(* ToolTens force +,++,-,-- *)
	IF xToolTensForceAdd OR xToolTensForceAddMore OR xToolTensForceSub OR xToolTensForceSubMore THEN
		CASE iStepAction OF
		(* check cylinder state *)
		1:	xTmp:=	ptrCylAction^.T_CtrleCyl.xDone
					AND NOT(ptrCylAction^.T_CtrleCyl.xExecute)
					AND NOT(ptrCylAction^.T_CtrleCyl.xErr)
					AND ptrCylAction^.T_CtrleCyl.T_AnalogCylinder.xActiv;
			(* next step *)
			IF xTmp THEN iStepAction:=10; ELSE iStepAction:=95; END_IF
			IF xTmp AND T_Station.TControl.xHardwareConfigError THEN iStepAction:=95; END_IF;
		10:	IF xToolTensForceAdd THEN
				rCorrectionValue:=0.1;
			END_IF;
			IF xToolTensForceAddMore THEN
				rCorrectionValue:=1.0;
			END_IF;
			IF xToolTensForceSub THEN
				rCorrectionValue:=-0.1;
			END_IF;
			IF xToolTensForceSubMore THEN
				rCorrectionValue:=-1.0;
			END_IF;
			T_Visu.ptrT_ExchgParam^.T_InfoValueCommon.rToolTensionForce:=T_Visu.ptrT_ExchgParam^.T_InfoValueCommon.rToolTensionForce + rCorrectionValue;
			IF (T_Visu.ptrT_ExchgParam^.T_InfoValueCommon.rToolTensionForce < 0.1) THEN
				T_Visu.ptrT_ExchgParam^.T_InfoValueCommon.rToolTensionForce:=0.0;
			END_IF;
			IF (T_Visu.ptrT_ExchgParam^.T_InfoValueCommon.rToolTensionForce > T_NovRAM.T_Data.T_Standard.T_ToolTensionSystem.rMaxForceTT) THEN
				T_Visu.ptrT_ExchgParam^.T_InfoValueCommon.rToolTensionForce:=T_NovRAM.T_Data.T_Standard.T_ToolTensionSystem.rMaxForceTT;
			END_IF;
			(* next step *)
			iStepAction:=20;
		(* activ function set analog value *)
		20:	ptrCylAction^.T_CtrleCyl.T_AnalogCylinder.rForceIn:=T_Visu.ptrT_ExchgParam^.T_InfoValueCommon.rToolTensionForce;
			ptrCylAction^.T_CtrleCyl.iFunction:=4;
			ptrCylAction^.T_CtrleCyl.xExecute:=TRUE;
			(* next step *)
			iStepAction:=30;
			xStepActionDone:=FALSE;
		(* wait confirmation *)
		30:	IF NOT(xStepActionDone) THEN
			(* release execution *)
				ptrCylAction^.T_CtrleCyl.xExecute:=FALSE;
				xStepActionDone:=TRUE;
			ELSE
				IF ptrCylAction^.T_CtrleCyl.xDone THEN
				(* action done *)
					iStepAction:=90;
					xStepActionDone:=FALSE;
				ELSE 	IF ptrCylAction^.T_CtrleCyl.xErr THEN
						(* action error *)
							iStepAction:=99;
							xStepActionDone:=FALSE;
						END_IF
				END_IF
			END_IF
		(* waiting time out *)
		89:	IF TimerAction.Q THEN iStepAction:=90; END_IF
		(* action done *)
		90:	T_Visu.T_CtrleAction.xDone:=TRUE;
			T_Visu.T_CtrleAction.xNotReady:=FALSE;
			T_Visu.T_CtrleAction.xErr:=FALSE;
			T_Visu.T_CtrleAction.udiErrorID:=0;
			xToolTensForceAdd:=xToolTensForceAddMore:=xToolTensForceSub:=xToolTensForceSubMore:=FALSE;
		(* cylinder not ready *)
		95:	TimerNotReady(IN:=TRUE);
			xToolTensForceAdd:=xToolTensForceAddMore:=xToolTensForceSub:=xToolTensForceSubMore:=FALSE;
		(* error *)
		99:	T_Visu.T_CtrleAction.xDone:=TRUE;
			T_Visu.T_CtrleAction.xNotReady:=FALSE;
			(*diErrorNr:=6000000 * ptrCylAction^.T_CtrleCyl.udiErrorID;*)
			diErrorNr:=9000000+ (1000000 * iSelectedCylinder) + ptrCylAction^.T_CtrleCyl.udiErrorID;
			FBErrorMessage(	diErrorNr:=diErrorNr,
							T_ErrorList:=T_ErrorList);
			T_Visu.ptrT_ExchgParam^.T_Visu.T_Message.sDynamicTextEnglish:=FBErrorMessage.sErrorTextEnglish;
			T_Visu.ptrT_ExchgParam^.T_Visu.T_Message.sDynamicTextDeutsch:=FBErrorMessage.sErrorTextDeutsch;
			T_Visu.ptrT_ExchgParam^.T_Visu.T_Message.sDynamicTextFrancais:=FBErrorMessage.sErrorTextFrancais;
			T_Visu.ptrT_ExchgParam^.T_SafetyCtrl.xSetForceError:=TRUE;
			T_Visu.ptrT_ExchgParam^.T_SafetyCtrl.diSetForceErrorNr:=diErrorNr;
			T_Visu.T_CtrleAction.xErr:=FALSE;
			T_Visu.T_CtrleAction.udiErrorID:=0;
			ptrCylAction^.T_CtrleCyl.xReset:=TRUE;
			xToolTensForceAdd:=xToolTensForceAddMore:=xToolTensForceSub:=xToolTensForceSubMore:=FALSE;
		END_CASE
	END_IF;
END_ACTION
ACTION VisuFunction_NovRAM:
(* Action Save NovRAM *)
	IF xAction_SaveNovRAM OR xAction_SaveNovRAMWithoutConfirm THEN
		(* Step saving NovRAM *)
		CASE iStepActionNovRam OF
		(* check NovRAM *)
		1:	xTmp:=	T_NovRAM.T_Ctrle.xDone
					AND NOT(T_NovRAM.T_Ctrle.xExecute)
					AND NOT(T_NovRAM.T_Ctrle.xErr);
			IF xTmp THEN
				(* next Step *)
				iStepActionNovRam :=10;
				xStepActionDone:=FALSE;
			(* activ error *)
			ELSE iStepActionNovRam:=95; END_IF
		(* copy value *)
		10:	IF  xAction_SaveNovRAM THEN
				(* saving with confirmation *)
				TimerAction(IN:=FALSE);
				tTimeOutAction:=T#6s;
				T_Visu.ptrT_ExchgParam^.T_Visu.T_Message.iState:=108;	(* Confirm saving action <Enter>, or escape <Esc> ? *)
				(* next Step *)
				iStepActionNovRam :=20;
			ELSE
				(* next Step *)
				IF xAction_LoadProfileToProcessImage OR xAction_SaveProfileToFile OR xActionDeleteProfile  THEN
					IF xAction_LoadProfileToProcessImage THEN
						T_NovRam.T_Data.T_Standard.T_InfoProcess.iProfile:=T_VisuQVis.ptrT_ExchgParam^.T_StationCommon.T_InfoProcess.iProfile;
						T_NovRam.T_Data.T_Standard.T_InfoProcess.sProfileName:=T_VisuQVis.ptrT_ExchgParam^.T_StationCommon.T_InfoProcess.sProfileName;
					END_IF;
					iStepActionNovRam :=40;
				ELSE
					iStepActionNovRam :=30;
				END_IF;
				(* Display message *)
				T_Visu.ptrT_ExchgParam^.T_Visu.T_Message.iState:=13;	(* Start saving *)
			END_IF;
		(* waiting for saving confirmation key <Enter> or <Esc> *)
		20:	IF RisingEdgeKeyPanel_Enter.Q THEN
			(* Display message *)
				T_Visu.ptrT_ExchgParam^.T_Visu.T_Message.iState:=13;	(* Start saving *)
				(* next step *)
				iStepActionNovRam:=30;
			ELSE
				IF RisingEdgeKeyPanel_Esc.Q THEN iStepActionNovRam:=60; END_IF
				(* An other message has been displayed, stop saving action *)
				IF T_Visu.ptrT_ExchgParam^.T_Visu.T_Message.iState<>108 THEN iStepActionNovRam:=60; END_IF
			END_IF
		30:	T_NovRAM.T_Data.T_ProcessImageData.T_GeometryPara:=T_Visu.ptrT_ExchgParam^.T_GeometryCommon.T_Geometry;
			T_NovRAM.T_Data.T_ProcessImageData.T_PrismPara:=T_Visu.ptrT_ExchgParam^.T_StationCommon.T_PrismPara;
			IF (T_NovRAM.T_Data.T_ProcessImageData.T_PrismPara.bStateInputPrisma = 1) THEN
				T_NovRAM.T_Data.T_ProcessImageData.T_PrismPara.bStateInputPrisma:=0;
			END_IF;
			IF (T_NovRAM.T_Data.T_ProcessImageData.T_PrismPara.bStateInputPrisma = 3) THEN
				T_NovRAM.T_Data.T_ProcessImageData.T_PrismPara.bStateInputPrisma:=2;
			END_IF;
			rCalcMinMaxToolDia:=	rFctCalcMaxToolDiameter(	rDistanceD1:=T_NovRAM.T_Data.T_ProcessImageData.T_PrismPara.rPrismaDistanceD1,
														rDistanceD2:=T_NovRAM.T_Data.T_ProcessImageData.T_PrismPara.rPrismaDistanceD2,
														rAnglePrism:=T_NovRAM.T_Data.T_ProcessImageData.T_PrismPara.rPrismaAngleA);
			T_NovRAM.T_Data.T_ProcessImageData.T_PrismPara.rToolDiameterMax:=rCalcMinMaxToolDia;
			rCalcMinMaxToolDia:=	rFctCalcMinToolDiameter(	rDistanceD1:=T_NovRAM.T_Data.T_ProcessImageData.T_PrismPara.rPrismaDistanceD1,
														rDistanceD2:=T_NovRAM.T_Data.T_ProcessImageData.T_PrismPara.rPrismaDistanceD2,
														rAnglePrism:=T_NovRAM.T_Data.T_ProcessImageData.T_PrismPara.rPrismaAngleA,
														bStateInputPrisma:=T_NovRAM.T_Data.T_ProcessImageData.T_PrismPara.bStateInputPrisma);
			T_NovRAM.T_Data.T_ProcessImageData.T_PrismPara.rToolDiameterMin:=rCalcMinMaxToolDia;
			rCalcPrismaFactor:=	rFctCalcPrismaFactor(	rAnglePrism:=T_NovRAM.T_Data.T_ProcessImageData.T_PrismPara.rPrismaAngleA);
			T_NovRAM.T_Data.T_ProcessImageData.T_PrismPara.rPrismaFactor:=rCalcPrismaFactor;
			T_Visu.ptrT_ExchgParam^.T_StationCommon.T_PrismPara:=T_NovRAM.T_Data.T_ProcessImageData.T_PrismPara;
			T_NovRAM.T_Data.T_Standard.T_TeachINToolLeft:=T_Visu.ptrT_ExchgParam^.T_TeachIn.TParam_ToolLeft;
			T_NovRAM.T_Data.T_Standard.T_TeachINToolCenter:=T_Visu.ptrT_ExchgParam^.T_TeachIn.TParam_ToolCenter;
			T_NovRAM.T_Data.T_Standard.T_TeachINToolRight:=T_Visu.ptrT_ExchgParam^.T_TeachIn.TParam_ToolRight;
			T_NovRAM.T_Data.T_Standard.T_TeachINToolFeeder:=T_Visu.ptrT_ExchgParam^.T_TeachIn.TParam_ToolFeeder;
			T_NovRAM.T_Data.T_Standard.T_TeachINGrindFeeder:=T_Visu.ptrT_ExchgParam^.T_TeachIn.TParam_GrindFeeder;
			T_NovRAM.T_Data.T_Standard.T_AxisPosition:=T_Visu.ptrT_ExchgParam^.T_TeachIn.TParam_AxisPosition;
			T_NovRAM.T_Data.T_Standard.T_MachineConfig.iConfigMachineType:=T_Visu.ptrT_ExchgParam^.T_StationCommon.iConfigMachineType;
			T_NovRAM.T_Data.T_Standard.T_MachineConfig.iConfigAxisType:=T_Visu.ptrT_ExchgParam^.T_StationCommon.iConfigAxisType;
			T_NovRAM.T_Data.T_Standard.T_MachineConfig.iConfigVisuNavigation:=T_Visu.ptrT_ExchgParam^.T_StationCommon.iConfigVisuNavigation;
			T_NovRAM.T_Data.T_Standard.T_MachineConfig.rConfigMaxToolLength:=T_Visu.ptrT_ExchgParam^.T_StationCommon.rConfigMaxToolLength;
			T_NovRAM.T_Data.T_Standard.T_ToolTensionSystem:=T_Visu.ptrT_ExchgParam^.T_StationCommon.T_ParamToolTensionSystem;
			T_NovRAM.T_Data.T_Standard.T_Cyl_ToolTension:=T_Visu.ptrT_ExchgParam^.T_Cylinder.T_ParamToolTension;
			T_NovRAM.T_Data.T_ProcessImageData.T_AutoGeometryPara:=T_Visu.ptrT_ExchgParam^.T_StationCommon.T_AutoGeometryPara;
			T_NovRAM.T_Data.T_ProcessImageData.T_AutoGroovePara:=T_Visu.ptrT_ExchgParam^.T_StationCommon.T_AutoGroovePara;
			T_NovRAM.T_Data.T_ProcessImageData.T_CalibrationPara:=T_Visu.ptrT_ExchgParam^.T_StationCommon.T_CalibrationPara;
			T_NovRAM.T_Data.T_ProcessImageData.T_ProcessPara:=T_Visu.ptrT_ExchgParam^.T_StationCommon.T_ProcessPara;
			T_NovRam.T_Data.TWarmUp_Para:=T_ExchgParam.T_FunctionCommon.TWarmUp_Para; (* SOA 21.02.2023*)
			(* next Step *)
			iStepActionNovRam :=40;
		(* activ save *)
		40:	T_NovRAM.T_Ctrle.xExecute:=TRUE;
			T_NovRAM.T_Ctrle.iFunction:=2;
			(* next Step *)
			iStepActionNovRam :=50;
			xStepActionDone:=FALSE;
		(* wait save confirmation *)
		50:	IF NOT(xStepActionDone) THEN
				T_NovRAM.T_Ctrle.xExecute:=FALSE;
				(* confirm Step *)
				xStepActionDone:=TRUE;
			ELSE
				IF T_NovRAM.T_Ctrle.xDone THEN
				(* next Step *)
					IF (T_Visu.T_PlcParam.dwActualPage = 430) OR ((T_Visu.T_PlcParam.dwActualPage = 130) AND (T_Visu.T_CtrleAction.iFunction = 1002)) OR
					     ((T_Visu.T_PlcParam.dwActualPage = 470) AND (T_Visu.ptrT_ExchgParam^.T_Config.iEditParam = 410)) THEN
						iStepActionNovRam :=51;
						xOpenMessageBox:=FALSE;
					ELSE
						iStepActionNovRam :=90;
					END_IF;
					xStepActionDone:=FALSE;
				ELSE	IF T_NovRAM.T_Ctrle.xErr THEN
							iStepActionNovRam:=99;
							xStepActionDone:=FALSE;
						END_IF
				END_IF
			END_IF
		(* check first if the Actual position is between the pos and neg SW limit switch *)
		51:	IF (T_Station.THardware.TAxisGrindFeeder.T_LiveValue.lrActualPosition >= T_NovRAM.T_Data.T_ProcessImageData.T_PrismPara.rToolDiameterMin) AND
			     (T_Station.THardware.TAxisGrindFeeder.T_LiveValue.lrActualPosition <= (T_NovRAM.T_Data.T_ProcessImageData.T_PrismPara.rToolDiameterMax + T_NovRAM.T_Data.T_Standard.T_TeachINGrindFeeder.rOffsetSWPosEndSwitch)) THEN
				(* Actual Position is not over the SW limit switches *)
				iStepActionNovRam :=53;
			ELSE
				(* Actual Position is over the SW limit switches *)
				T_Station.THardware.TAxisGrindFeeder.T_CtrleSingle.iFunction:=29;		(* Switch off the SW limit switches, in this case the GrindFeeder will not move automatically *)
				T_Station.THardware.TAxisGrindFeeder.T_CtrleSingle.xExecute:=TRUE;
				iStepActionNovRam :=52;
				xOpenMessageBox:=TRUE;
				tTimeOutAction:=tTimeOutAction + T#9999s;
			END_IF;
		(* Wait end of resettet SW end switch for the GrindFeeder Axis *)
		52:	IF NOT(T_Station.THardware.TAxisGrindFeeder.T_CtrleSingle.xExecute) AND T_Station.THardware.TAxisGrindFeeder.T_CtrleSingle.xDone THEN
				(* set the new position of the GrindFeeder Axis *)
				T_Station.THardware.TAxisGrindFeeder.T_CtrleSingle.rSetPosition:=T_NovRAM.T_Data.T_ProcessImageData.T_PrismPara.rToolDiameterMin;
				T_Station.THardware.TAxisGrindFeeder.T_CtrleSingle.iFunction:=11;
				T_Station.THardware.TAxisGrindFeeder.T_CtrleSingle.xExecute:=TRUE;
				lrActualGrindFeedPosition:=DINT_TO_LREAL(LREAL_TO_DINT(T_Station.THardware.TAxisGrindFeeder.T_LiveValue.lrActualPosition * 100.0)) / 100.0;
				lrToWriteGrindFeedPosition:=DINT_TO_LREAL(LREAL_TO_DINT(T_NovRAM.T_Data.T_ProcessImageData.T_PrismPara.rToolDiameterMin * 100.0)) / 100.0;
				iStepActionNovRam :=53;
			END_IF;
			IF NOT(T_Station.THardware.TAxisGrindFeeder.T_CtrleSingle.xExecute) AND T_Station.THardware.TAxisGrindFeeder.T_CtrleSingle.xErr THEN
				iStepActionNovRam :=98;
			END_IF;
		(* Set SW end switch for the GrindFeeder Axis *)
		53:	IF NOT(T_Station.THardware.TAxisGrindFeeder.T_CtrleSingle.xExecute) AND T_Station.THardware.TAxisGrindFeeder.T_CtrleSingle.xDone THEN
				T_Station.THardware.TAxisGrindFeeder.T_CtrleSingle.iFunction:=28;
				T_Station.THardware.TAxisGrindFeeder.T_CtrleSingle.lrSWNegLimitSwitch:=T_NovRAM.T_Data.T_ProcessImageData.T_PrismPara.rToolDiameterMin;
				T_Station.THardware.TAxisGrindFeeder.T_CtrleSingle.lrSWPosLimitSwitch:=T_NovRAM.T_Data.T_ProcessImageData.T_PrismPara.rToolDiameterMax + T_NovRAM.T_Data.T_Standard.T_TeachINGrindFeeder.rOffsetSWPosEndSwitch;
				T_Station.THardware.TAxisGrindFeeder.T_CtrleSingle.xExecute:=TRUE;
				iStepActionNovRam :=54;
			END_IF;
			IF NOT(T_Station.THardware.TAxisGrindFeeder.T_CtrleSingle.xExecute) AND T_Station.THardware.TAxisGrindFeeder.T_CtrleSingle.xErr THEN
				iStepActionNovRam :=98;
			END_IF;
		(* Wait end of settled SW end switch for the GrindFeeder Axis *)
		54:	IF NOT(T_Station.THardware.TAxisGrindFeeder.T_CtrleSingle.xExecute) AND T_Station.THardware.TAxisGrindFeeder.T_CtrleSingle.xDone THEN
				IF xOpenMessageBox THEN
					xOpenMessageBox:=FALSE;
					iStepActionNovRam :=55;
				ELSE
					iStepActionNovRam :=90;
				END_IF;
			END_IF;
			IF NOT(T_Station.THardware.TAxisGrindFeeder.T_CtrleSingle.xExecute) AND T_Station.THardware.TAxisGrindFeeder.T_CtrleSingle.xErr THEN
				iStepActionNovRam :=98;
			END_IF;
		(* Open MessageBox *)
		55:	T_Visu.ptrT_ExchgParam^.T_FunctionCommon.sMessageBoxLine1:='The prisma value are changed and the actual ';
			T_Visu.ptrT_ExchgParam^.T_FunctionCommon.sMessageBoxLine2:='GrindFeeder position is now over the';
			T_Visu.ptrT_ExchgParam^.T_FunctionCommon.sMessageBoxLine3:='Software limit switches. The actual absolut';
			T_Visu.ptrT_ExchgParam^.T_FunctionCommon.sMessageBoxLine4:='GrindFeeder position: ';
			T_Visu.ptrT_ExchgParam^.T_FunctionCommon.sMessageBoxLine4:=CONCAT(T_Visu.ptrT_ExchgParam^.T_FunctionCommon.sMessageBoxLine4,
																				LREAL_TO_STRING(lrActualGrindFeedPosition));
			T_Visu.ptrT_ExchgParam^.T_FunctionCommon.sMessageBoxLine4:=CONCAT(T_Visu.ptrT_ExchgParam^.T_FunctionCommon.sMessageBoxLine4,'um');
			T_Visu.ptrT_ExchgParam^.T_FunctionCommon.sMessageBoxLine5:='is overwritten with the minimum ';
			T_Visu.ptrT_ExchgParam^.T_FunctionCommon.sMessageBoxLine6:='ToolDiameter: ';
			T_Visu.ptrT_ExchgParam^.T_FunctionCommon.sMessageBoxLine6:=CONCAT(T_Visu.ptrT_ExchgParam^.T_FunctionCommon.sMessageBoxLine6,
																				LREAL_TO_STRING(lrToWriteGrindFeedPosition));
			T_Visu.ptrT_ExchgParam^.T_FunctionCommon.sMessageBoxLine6:=CONCAT(T_Visu.ptrT_ExchgParam^.T_FunctionCommon.sMessageBoxLine6,'um');
			T_Visu.ptrT_ExchgParam^.T_FunctionCommon.xOpenOverlayMessageBox:=TRUE;
			iStepActionNovRam :=56;
		(* Wait cofirming of the messagebox *)
		56:	IF NOT(T_Visu.ptrT_ExchgParam^.T_FunctionCommon.xOpenOverlayMessageBox) THEN
				iStepActionNovRam :=90;
			END_IF;
			IF T_Visu.T_CtrleAction.xDone THEN
				T_Visu.ptrT_ExchgParam^.T_FunctionCommon.xOpenOverlayMessageBox:=FALSE;
				xAction_SaveNovRAM:=FALSE;
				xAction_SaveNovRAMWithoutConfirm:=FALSE;
				T_Visu.ptrT_ExchgParam^.T_Visu.T_Message.iState:=0;
			END_IF;
		(* Reset settled value *)
		60:	xResetParaListValue:=TRUE;
			iStepActionNovRam:=70;
		70:	IF NOT(xResetParaListValue) THEN
				iStepActionNovRam:=90;
			END_IF;
		(* no code, waiting timeout *)
		89:	IF TimerAction.Q THEN iStepActionNovRam:=90; END_IF
		(* save done *)
		90:	T_Visu.ptrT_ExchgParam^.T_Visu.T_Message.iState:=0;
			T_Visu.T_CtrleAction.xDone:=TRUE;
			T_Visu.T_CtrleAction.xNotReady:=FALSE;
			T_Visu.T_CtrleAction.xErr:=FALSE;
			T_Visu.T_CtrleAction.udiErrorID:=0;
			xAction_SaveNovRAM:=FALSE;
			xAction_SaveNovRAMWithoutConfirm:=FALSE;
			T_Visu.ptrT_ExchgParam^.T_FunctionCommon.xOpenOverlayMessageBox:=FALSE;
		(* NovRAM not ready *)
		95:	TimerNotReady(IN:=TRUE);
			xAction_SaveNovRAM:=FALSE;
			xAction_SaveNovRAMWithoutConfirm:=FALSE;
			T_Visu.ptrT_ExchgParam^.T_FunctionCommon.xOpenOverlayMessageBox:=FALSE;
		(* error *)
		98:	T_Visu.ptrT_ExchgParam^.T_StationCommon.wState:=T_Visu.ptrT_ExchgParam^.T_StationCommon.wState AND 16#BF;
			T_Visu.T_CtrleAction.xDone:=TRUE;
			T_Visu.T_CtrleAction.xNotReady:=FALSE;
			IF (T_Station.THardware.TAxisGrindFeeder.T_Config_Gen.iTyp <> 0) THEN
				diErrorNr:=(T_Station.THardware.TAxisGrindFeeder.T_Config_Gen.iTyp * 1000000) + T_Station.THardware.TAxisGrindFeeder.T_CtrleSingle.udiErrorID;
			ELSE
				diErrorNr:=0;
			END_IF;
			FBErrorMessage(	diErrorNr:=diErrorNr,
							T_ErrorList:=T_ErrorList);
			T_Visu.ptrT_ExchgParam^.T_Visu.T_Message.sDynamicTextEnglish:=FBErrorMessage.sErrorTextEnglish;
			T_Visu.ptrT_ExchgParam^.T_Visu.T_Message.sDynamicTextDeutsch:=FBErrorMessage.sErrorTextDeutsch;
			T_Visu.ptrT_ExchgParam^.T_Visu.T_Message.sDynamicTextFrancais:=FBErrorMessage.sErrorTextFrancais;
			T_Visu.ptrT_ExchgParam^.T_SafetyCtrl.xSetForceError:=TRUE;
			T_Visu.ptrT_ExchgParam^.T_SafetyCtrl.diSetForceErrorNr:=diErrorNr;
			T_Visu.T_CtrleAction.xErr:=FALSE;
			T_Visu.T_CtrleAction.udiErrorID:=0;
			T_Station.THardware.TAxisGrindFeeder.T_CtrleSingle.iFunction:=1;
			T_Station.THardware.TAxisGrindFeeder.T_CtrleSingle.xExecute:=TRUE;
			xAction_SaveNovRAM:=FALSE;
			xAction_SaveNovRAMWithoutConfirm:=FALSE;
			T_Visu.ptrT_ExchgParam^.T_FunctionCommon.xOpenOverlayMessageBox:=FALSE;
		(* error *)
		99:	T_Visu.T_CtrleAction.xDone:=FALSE;
			T_Visu.T_CtrleAction.xNotReady:=FALSE;
			T_Visu.T_CtrleAction.xErr:=TRUE;
			T_Visu.T_CtrleAction.udiErrorID:=16#F0000 + T_Visu.T_CtrleAction.iFunction;
			xAction_SaveNovRAM:=FALSE;
			xAction_SaveNovRAMWithoutConfirm:=FALSE;
			T_Visu.ptrT_ExchgParam^.T_FunctionCommon.xOpenOverlayMessageBox:=FALSE;
		END_CASE
	END_IF;
END_ACTION
ACTION VisuFunction_ProcessFunction:
(* Action start process machine or station *)
	IF xActionProcMachine OR xActionProcStation THEN
		(* Step process machine *)
		CASE iStepAction OF
		(* check process state *)
		1:	xTmp:=	T_Process.xEnable AND
					T_Process.xEnd AND
					T_Process.xRdy AND
					NOT(T_Process.xStop) AND
					NOT(T_Process.xStopCycle) AND
					NOT(T_Process.xError);
			(* next step *)
			IF NOT(xTmp) THEN
				iStepAction:=95;
			ELSE IF xActionProcMachine THEN iStepAction:=10; ELSE iStepAction:=20; END_IF
			END_IF
		(* check process number and start process machine *)
		10:	CASE T_Process.iFunctNr OF
			(* process available *)
			(*	10=Process AutoGeometry
				20=Process AutoGroove
				30=Process Reference
			*)
			10,20,30:	T_Visu.T_CtrleProcess.iFunction:=1;
						T_Visu.T_CtrleProcess.xExecute:=TRUE;
						iStepAction:=90;
			(* unknown process *)
			ELSE	iStepAction:=95;
			END_CASE
			(* next step *)
			xStepActionDone:=FALSE;
		(* check process number and start process station *)
		20:	CASE T_Process.iFunctNr OF
			(* process available *)
			(*	40=ToolCalibration
			*)
			40:	T_Visu.T_CtrleProcess.iFunction:=2;
				T_Visu.T_CtrleProcess.xExecute:=TRUE;
				iStepAction:=90;
			(* unknown process *)
			ELSE
				iStepAction:=95;
			END_CASE
			(* next step *)
			xStepActionDone:=FALSE;
		(* Display message, waiting timeout *)
		89:	IF TimerAction.Q THEN
				(* init. trigger FB_CtrleButton Start/Stop *)
				T_Visu.ptrT_ExchgParam^.T_Machine.T_Process.wState:=16#0;
				(* action done *)
				iStepAction:=90;
			END_IF
		(* action done *)
		90:	T_Visu.T_CtrleAction.xDone:=TRUE;
			T_Visu.T_CtrleAction.xNotReady:=FALSE;
			T_Visu.T_CtrleAction.xErr:=FALSE;
			T_Visu.T_CtrleAction.udiErrorID:=0;
			xActionProcMachine:=FALSE;
			xActionProcStation:=FALSE;
		(* cylinder not ready *)
		95:	TimerNotReady(IN:=TRUE);
			xActionProcMachine:=FALSE;
			xActionProcStation:=FALSE;
		(* error *)
		99:	T_Visu.T_CtrleAction.xDone:=FALSE;
			T_Visu.T_CtrleAction.xNotReady:=FALSE;
			T_Visu.T_CtrleAction.xErr:=TRUE;
			T_Visu.T_CtrleAction.udiErrorID:=16#F0000 + T_Visu.T_CtrleAction.iFunction;
			xActionProcMachine:=FALSE;
			xActionProcStation:=FALSE;
		END_CASE
	END_IF
END_ACTION
ACTION VisuFunction_ProcessStop:
(* Stop process *)
	IF xStopProcess OR xAction_StopCycle THEN
		(* Set stop process *)
		CASE iStepAction OF
		(* check process state and stop process if possible *)
		1:	IF NOT xStopButton THEN
				xTmp:=	T_Process.xRdy
						AND NOT T_Process.xStop
						AND NOT T_Process.xStopCycle
						AND NOT T_Process.xEnd
						AND NOT T_Process.xError
						AND NOT T_Process.xAbord;
				IF xStopProcess AND T_Process.xStopCycle AND NOT(T_Process.xEnd) AND NOT(T_Process.xError) AND NOT(T_Process.xStop) THEN
					xTmp:=TRUE;
				END_IF;
				IF xAction_StopCycle THEN
					IF (T_NovRAM.T_Data.T_ProcessImageData.T_AutoGeometryPara.iCycleGeometry <= 1) THEN
						xTmp:=FALSE;
					END_IF;
				END_IF;
				IF xTmp THEN
					IF xStopProcess THEN
					(* activ stop immediat *)
						T_Process.xStop:=TRUE;
						T_Process.xStopCycle:=NOT T_Process.xStop;
						xBlockConfirmMessage:=TRUE;
						(* Display info message *)
						T_Visu.ptrT_ExchgParam^.T_Visu.T_Message.iState:=122;	(* Stop process immediately *)
						(* set variable *)
						xStopImmediatly:=TRUE;
						(* next step *)
						iStepAction:=20;
					END_IF;
					IF xAction_StopCycle THEN
						T_Process.xStopCycle:=TRUE;
						T_Process.xStop:=NOT T_Process.xStopCycle;
						xBlockConfirmMessage:=TRUE;
						(* Display message *)
						T_Visu.ptrT_ExchgParam^.T_Visu.T_Message.iState:=103;	(* Process will be stopped at the end of the cycle *)
						(* next step *)
						iStepAction:=20;
					END_IF;
				(* not ready to execute stop *)
				ELSE iStepAction:=95; END_IF
			END_IF
			IF T_Process.xError THEN iStepAction:=99; END_IF
		(* waiting function done *)
		20:	IF T_Visu.T_CtrleVisu.xDone THEN
				IF (T_Visu.T_PlcParam.dwActualPage = 10) OR (T_Visu.T_PlcParam.dwActualPage = 20) OR (T_Visu.T_PlcParam.dwActualPage = 30) OR (T_Visu.T_PlcParam.dwActualPage = 110) THEN
					xWaitStopEnd:=xStopProcess;
					xWaitStopCycleEnd:=xAction_StopCycle;
					iStepWaitStopEnd:=1;
				ELSE
					xWaitStopEnd:=FALSE;
					xWaitStopCycleEnd:=FALSE;
				END_IF;
				(* no activ station for machine level *)
				IF T_Visu.T_PlcParam.dwActualPage < 100 THEN
					T_Visu.ptrT_ExchgParam^.T_TouchScreenBtPanel.iStateBtLeft:=0;
				END_IF
				(* next step *)
				iStepAction:=90;
			END_IF
			IF T_Visu.T_CtrleVisu.xErr THEN iStepAction:=99; END_IF
		(* End function *)
		90:	T_Visu.T_CtrleAction.xDone:=TRUE;
			T_Visu.T_CtrleAction.xErr:=FALSE;
			T_Visu.T_CtrleAction.udiErrorID:=16#0;
			xStopProcess:=FALSE;
			xAction_StopCycle:=FALSE;
		(* not ready *)
		95:	TimerNotReady(IN:=TRUE);
			xStopProcess:=FALSE;
			xAction_StopCycle:=FALSE;
		(* Error *)
		99:	T_Visu.T_CtrleAction.xDone:=FALSE;
			T_Visu.T_CtrleAction.xErr:=TRUE;
			T_Visu.T_CtrleAction.udiErrorID:=16#F0000 + T_Visu.T_CtrleAction.iFunction;
			xStopProcess:=FALSE;
			xAction_StopCycle:=FALSE;
		END_CASE
	END_IF

(* Wait End of Stop Machine Process *)
	IF xWaitStopEnd OR xWaitStopCycleEnd THEN
		CASE iStepWaitStopEnd OF
			1:	IF T_Process.xEnd THEN
					iStepWaitStopEnd:=10;
				END_IF;
				IF T_Process.xError THEN
					xWaitStopEnd:=FALSE;
					xWaitStopCycleEnd:=FALSE;
					iStepWaitStopEnd:=1;
				END_IF;
			10:	IF NOT(T_Visu.T_CtrleVisu.xExecute) AND T_Visu.T_CtrleVisu.xDone THEN
					T_Visu.ptrT_ExchgParam^.T_Visu.T_Message.iState:=0;
					IF (T_Process.iFunctNr = 30) THEN
						T_StartUp.T_Ctrle.xExecute:=TRUE;
						T_StartUp.T_Ctrle.iFunction:=11;	(* Acitvate Info Message Overlay *)
						(* THE REFERENCE DRIVE IS STOPPED! *)
						(* CONFIRM THIS MESSAGE AND *)
						(* THE MACHINE WILL BE READY! *)
						(*  *)
						T_StartUp.T_Ctrle.iMsgNumber:=5;
					END_IF;
					IF (T_Process.iFunctNr = 10) OR (T_Process.iFunctNr = 20) THEN
						T_StartUp.T_Ctrle.xExecute:=TRUE;
						T_StartUp.T_Ctrle.iFunction:=11;	(* Acitvate Info Message Overlay *)
						(* THE AUTO MODE CYCLE IS STOPPED! *)
						(* CONFIRM THIS MESSAGE AND *)
						(* THE MACHINE WILL BE READY! *)
						(*  *)
						T_StartUp.T_Ctrle.iMsgNumber:=4;
					END_IF;
					xWaitStopEnd:=FALSE;
					xWaitStopCycleEnd:=FALSE;
					iStepWaitStopEnd:=1;
				END_IF;
		END_CASE;
	END_IF;
END_ACTION
ACTION VisuFunction_ProfileManagement:
(* Copy profile value to process *)
	IF xAction_CopyProfileToProcess THEN
		(* Set copy action *)
		CASE iStepAction OF
		(* Set default value *)
		1:	(*IF xFctSetDefaultValueProfileOnlineChange(ptrNovRAM:=ADR(T_WorkingData),
												   ptrDefaultProfilStandProcPara:=ADR(T_DefaultProfilStandProcPara),
												   bActiveStation:=0) THEN iStepAction:=5; END_IF*)
			iStepAction:=10;
			(* Init. display value *)
			xProfileFileNotFound:=FALSE;
		(* activ reading profile file *)
		10:	IF (T_Visu.ptrT_ExchgParam^.T_StationCommon.T_InfoProcess.iProfile > 0) AND (T_Visu.ptrT_ExchgParam^.T_StationCommon.T_InfoProcess.iProfile <= csiMaxProfile) THEN
				T_Profile.T_Id.iNumber:=T_Visu.ptrT_ExchgParam^.T_StationCommon.T_InfoProcess.iProfile;
				T_Profile.T_Id.sName:=T_Visu.ptrT_ExchgParam^.T_StationCommon.T_InfoProcess.sProfileName;
				T_Profile.T_Ctrle.iFunction:=1;
				T_Profile.T_Ctrle.xExecute:=TRUE;
				(* next step *)
				iStepAction:=20;
			ELSE iStepAction:=25; END_IF
		20:	IF NOT T_Profile.T_Ctrle.xExecute AND T_Profile.T_Ctrle.xDone THEN
				(* next step *)
				iStepAction:=90;
			END_IF
			IF T_Profile.T_Ctrle.xErr THEN
				xProfileFileNotFound:=TRUE;
				iToLoadProfileNr:=T_Profile.T_Id.iNumber;
				sToLoadProfileName:=T_Profile.T_Id.sName;
				(* activ reset *)
				T_Profile.T_Ctrle.xReset:=TRUE;
				(* next step *)
				iStepAction:=25;
			END_IF
		(* waiting flag *)
		25:	IF NOT T_Profile.T_Ctrle.xReset AND T_Profile.T_Ctrle.xDone THEN
				IF (T_Profile.T_Id.iNumber = 1) THEN
					(*T_ActualProfilStandProcPara[1]:=T_DefaultProfilStandProcPara[1];*)
					iStepAction:=90;
				ELSE
					iStepAction:=26;
				END_IF;
				(* erase name *)
				T_NovRam.T_Data.T_IDProfileStation[1].sName:='Default';
				T_NovRam.T_Data.T_IDProfileStation[1].iNumber:=1;
				T_Visu.ptrT_ExchgParam^.T_StationCommon.T_InfoProcess.sProfileName:='Default';
				T_Visu.ptrT_ExchgParam^.T_StationCommon.T_InfoProcess.iProfile:=1;
			END_IF
			IF T_Profile.T_Ctrle.xErr THEN iStepAction:=99; END_IF
		(* activ reading profile file *)
		26:	T_Profile.T_Id.iNumber:=1;
			T_Profile.T_Id.sName:='Default';
			T_Profile.T_Ctrle.iFunction:=1;
			T_Profile.T_Ctrle.xExecute:=TRUE;
			(* next step *)
			iStepAction:=20;
		(* End function *)
		90:	IF xProfileFileNotFound THEN
				xProfileFileNotFound:=FALSE;
				sTmpDynamicText:=INT_TO_STRING(iToLoadProfileNr);
				sTmpDynamicText:=CONCAT(sTmpDynamicText,' ');
				(* For English Language *)
				T_Visu.ptrT_ExchgParam^.T_Visu.T_Message.sDynamicTextEnglish:=CONCAT(T_ErrorList.asErrorListEnglish.T_LanguagList[50],sTmpDynamicText);	(* 'Profile file not found: ' *)
				T_Visu.ptrT_ExchgParam^.T_Visu.T_Message.sDynamicTextEnglish:=CONCAT(T_Visu.ptrT_ExchgParam^.T_Visu.T_Message.sDynamicTextEnglish,sToLoadProfileName);
				(* For German Language *)
				T_Visu.ptrT_ExchgParam^.T_Visu.T_Message.sDynamicTextDeutsch:=CONCAT(T_ErrorList.asErrorListDeutsch.T_LanguagList[50],sTmpDynamicText);	(* 'Profile file not found: ' *)
				T_Visu.ptrT_ExchgParam^.T_Visu.T_Message.sDynamicTextDeutsch:=CONCAT(T_Visu.ptrT_ExchgParam^.T_Visu.T_Message.sDynamicTextDeutsch,sToLoadProfileName);
				(* For French Language *)
				T_Visu.ptrT_ExchgParam^.T_Visu.T_Message.sDynamicTextFrancais:=CONCAT(T_ErrorList.asErrorListFrancais.T_LanguagList[50],sTmpDynamicText);	(* 'Profile file not found: ' *)
				T_Visu.ptrT_ExchgParam^.T_Visu.T_Message.sDynamicTextFrancais:=CONCAT(T_Visu.ptrT_ExchgParam^.T_Visu.T_Message.sDynamicTextFrancais,sToLoadProfileName);
				T_Visu.ptrT_ExchgParam^.T_SafetyCtrl.xSetForceError:=TRUE;
				T_Visu.ptrT_ExchgParam^.T_SafetyCtrl.diSetForceErrorNr:=1;	(* Datei für Profile nicht gefunden *)
			END_IF;
			xUpdateProfileList:=TRUE;
			T_Visu.T_CtrleAction.xDone:=TRUE;
			T_Visu.T_CtrleAction.xErr:=FALSE;
			T_Visu.T_CtrleAction.udiErrorID:=16#0;
			xAction_CopyProfileToProcess:=FALSE;
		(* not ready *)
		95:	TimerNotReady(IN:=TRUE);
			xAction_CopyProfileToProcess:=FALSE;
		(* Error *)
		99:	T_Visu.T_CtrleAction.xDone:=FALSE;
			T_Visu.T_CtrleAction.xErr:=TRUE;
			T_Visu.T_CtrleAction.udiErrorID:=16#F1000 + T_Profile.T_Ctrle.iFunction;
			xAction_CopyProfileToProcess:=FALSE;
		END_CASE
	END_IF

(* Load profile to process image *)
	IF xAction_LoadProfileToProcessImage THEN
		(* Step import/export profile value *)
		CASE iStepAction OF
		(* Display message to ask for confirmation *)
		1:	T_Visu.ptrT_ExchgParam^.T_Visu.T_Message.iState:=111;
			(* next step *)
			iStepAction:=10;
		(* waiting for key <Enter> or <Esc> *)
		10:	IF RisingEdgeKeyPanel_Enter.Q THEN
				xProfileFileNotFound:=FALSE;
				(* Display message transfering *)
				T_Visu.ptrT_ExchgParam^.T_Visu.T_Message.iState:=15;
				(* next step *)
				iStepAction:=20;
			ELSE
				IF RisingEdgeKeyPanel_Esc.Q THEN iStepAction:=90; END_IF
				(* An other message has been displayed, stop import/export action *)
				IF T_Visu.ptrT_ExchgParam^.T_Visu.T_Message.iState<>105 AND  T_Visu.ptrT_ExchgParam^.T_Visu.T_Message.iState<>111THEN iStepAction:=90; END_IF
			END_IF
		(* Init. reading profile file *)
		20:	IF T_NovRam.T_Data.T_IDProfileStation[T_Visu.ptrT_ExchgParam^.T_ProfileCommon.T_Id.iNumber].sName <> '' THEN
			(* Profile name exists *)
				T_Profile.T_Id.iNumber:=T_Visu.ptrT_ExchgParam^.T_ProfileCommon.T_Id.iNumber;
				T_Profile.T_Id.sName:=T_NovRam.T_Data.T_IDProfileStation[T_Visu.ptrT_ExchgParam^.T_ProfileCommon.T_Id.iNumber].sName;
				T_Profile.T_Ctrle.iFunction:=1;
				T_Profile.T_Ctrle.xExecute:=TRUE;
				(* Display info message *)
				T_Visu.ptrT_ExchgParam^.T_Visu.T_Message.iState:=15;
				(* next step *)
				iStepAction:=30;
			(* Display info message 'file does not exists *)
			ELSE
				T_Visu.ptrT_ExchgParam^.T_Visu.T_Message.iState:=11;
				(* next step *)
				iStepAction:=50;
				xStepActionDone:=FALSE;
				tTimeOutAction:=TimerAction.ET+T#2s;
			END_IF
		(* waiting confirmation signal *)
		30:	IF NOT T_Profile.T_Ctrle.xExecute AND T_Profile.T_Ctrle.xDone THEN
			(* Copy profile to online value *)
				T_NovRam.T_Data.T_ProcessImageData:=T_NovRam.T_Data.T_ProcessImageLoadData;
				xResetParaListValue:=TRUE;
				(* next step *)
				iStepAction:=60;
			END_IF
			IF T_Profile.T_Ctrle.xErr THEN
				IF T_Profile.T_Id.iNumber > 1 THEN
				(* Reset profile value, display message and reset profile error *)
					(*xFctResetProfileValue(ptrProfileData:=ADR(T_Profile.T_DataOnline));*)
					T_Visu.ptrT_ExchgParam^.T_ProfileCommon.T_Id.sName:='';
					(* Profile will be erased from the profile list *)
					T_NovRam.T_Data.T_IDProfileStation[T_Visu.ptrT_ExchgParam^.T_ProfileCommon.T_Id.iNumber].sName:='';
					xUpdateProfileList:=TRUE;
					(* Display info message 'file does not exists *)
					T_Visu.ptrT_ExchgParam^.T_Visu.T_Message.iState:=11;
					(* Reset control profile *)
					T_Profile.T_Ctrle.xReset:=TRUE;
					(* next step *)
					iStepAction:=40;
					xStepActionDone:=FALSE;
					(* use tmp timer to diplay message *)
					TimerONTmp(IN:=FALSE);
					TimerONTmp.PT:=T#1s;
				ELSE
					xProfileFileNotFound:=TRUE;
					iToLoadProfileNr:=1;
					sToLoadProfileName:='Default';
					(* Set Static Default Parameter *)
(*
					IF xFctSetDefaultValueProfileOnlineChange(ptrNovRAM:=ADR(T_WorkingData),
									ptrDefaultProfilStandProcPara:=ADR(T_DefaultProfilStandProcPara),
									bActiveStation:=T_Visu.ptrT_ExchgParam^.T_Visu.bActivStation) THEN
						T_WorkingData.T_Station[T_Visu.ptrT_ExchgParam^.T_Visu.bActivStation].T_StProcess:=T_DefaultProfilStandProcPara[T_Visu.ptrT_ExchgParam^.T_Visu.bActivStation];
						T_ActualProfilStandProcPara[T_Visu.ptrT_ExchgParam^.T_Visu.bActivStation]:=T_DefaultProfilStandProcPara[T_Visu.ptrT_ExchgParam^.T_Visu.bActivStation];
						T_Visu.ptrT_ExchgParam^.T_StationCommon.T_ParamStProcess:=T_DefaultProfilStandProcPara[T_Visu.ptrT_ExchgParam^.T_Visu.bActivStation];
						T_WorkingData.T_Station[T_Visu.ptrT_ExchgParam^.T_Visu.bActivStation].T_InfoProcess.iProfile:=1;
						T_WorkingData.T_Station[T_Visu.ptrT_ExchgParam^.T_Visu.bActivStation].T_Config.iProfile:=1;
						T_WorkingData.T_Station[T_Visu.ptrT_ExchgParam^.T_Visu.bActivStation].T_InfoProcess.sProfileName:='Default';
						T_Visu.ptrT_ExchgParam^.T_StationCommon.T_InfoProcess.iProfile:=1;
						T_Visu.ptrT_ExchgParam^.T_StationCommon.T_InfoProcess.sProfileName:='Default';
						(* Reset control profile *)
						T_Profile.T_Ctrle.xReset:=TRUE;
						(* next step *)
						iStepAction:=60;
					END_IF;
*)
				END_IF;
			END_IF
		(* Wait delay timer *)
		40:	IF TimerONTmp.Q THEN
				T_Visu.ptrT_ExchgParam^.T_Visu.T_Message.iState:=0;
				(* next step *)
				iStepAction:=60;
			END_IF
		(* delay time out *)
		50:	IF TimerAction.Q THEN xAction_LoadProfileToProcessImage:=FALSE; END_IF
		(* active saving data NovRAM *)
		60:	IF NOT(xResetParaListValue) THEN
				xAction_SaveNovRAMWithoutConfirm:=TRUE;
				iStepActionNovRam:=1;
				(* next step *)
				iStepAction:=80;
			END_IF;
		(* waiting confirm saving NovRAM action *)
		80:	IF NOT xAction_SaveNovRAMWithoutConfirm THEN
				iStepAction:=90;
			END_IF;
		(* save done *)
		90:	IF xProfileFileNotFound THEN
				xProfileFileNotFound:=FALSE;
				sTmpDynamicText:=INT_TO_STRING(iToLoadProfileNr);
				sTmpDynamicText:=CONCAT(sTmpDynamicText,' ');
				sTmpDynamicText:=CONCAT(sTmpDynamicText,sToLoadProfileName);
				(* For English Language *)
				T_Visu.ptrT_ExchgParam^.T_Visu.T_Message.sDynamicTextEnglish:=CONCAT(T_ErrorList.asErrorListEnglish.T_LanguagList[50],sTmpDynamicText);	(* 'Profile file not found: ' *)
				T_Visu.ptrT_ExchgParam^.T_Visu.T_Message.sDynamicTextEnglish:=CONCAT(T_Visu.ptrT_ExchgParam^.T_Visu.T_Message.sDynamicTextEnglish,T_ErrorList.asErrorListEnglish.T_LanguagList[51]);	(* ' -->Load static default parameter' *)
				(* For German Language *)
				T_Visu.ptrT_ExchgParam^.T_Visu.T_Message.sDynamicTextDeutsch:=CONCAT(T_ErrorList.asErrorListDeutsch.T_LanguagList[50],sTmpDynamicText);	(* 'Profile file not found: ' *)
				T_Visu.ptrT_ExchgParam^.T_Visu.T_Message.sDynamicTextDeutsch:=CONCAT(T_Visu.ptrT_ExchgParam^.T_Visu.T_Message.sDynamicTextDeutsch,T_ErrorList.asErrorListDeutsch.T_LanguagList[51]);	(* ' -->Load static default parameter' *)
				(* For French Language *)
				T_Visu.ptrT_ExchgParam^.T_Visu.T_Message.sDynamicTextFrancais:=CONCAT(T_ErrorList.asErrorListFrancais.T_LanguagList[50],sTmpDynamicText);	(* 'Profile file not found: ' *)
				T_Visu.ptrT_ExchgParam^.T_Visu.T_Message.sDynamicTextFrancais:=CONCAT(T_Visu.ptrT_ExchgParam^.T_Visu.T_Message.sDynamicTextFrancais,T_ErrorList.asErrorListFrancais.T_LanguagList[51]);	(* ' -->Load static default parameter' *)
				T_Visu.ptrT_ExchgParam^.T_SafetyCtrl.xSetForceError:=TRUE;
				T_Visu.ptrT_ExchgParam^.T_SafetyCtrl.diSetForceErrorNr:=1;	(* Datei für Profile nicht gefunden *)
			END_IF;
			T_Visu.ptrT_ExchgParam^.T_Visu.T_Message.iState:=0;
			T_Visu.T_CtrleAction.xDone:=TRUE;
			T_Visu.T_CtrleAction.xNotReady:=FALSE;
			T_Visu.T_CtrleAction.xErr:=FALSE;
			T_Visu.T_CtrleAction.udiErrorID:=0;
			xAction_LoadProfileToProcessImage:=FALSE;
		(* Action not ready *)
		95:	TimerNotReady(IN:=TRUE);
			xAction_LoadProfileToProcessImage:=FALSE;
		(* error *)
		99:	T_Visu.T_CtrleAction.xDone:=FALSE;
			T_Visu.T_CtrleAction.xNotReady:=FALSE;
			T_Visu.T_CtrleAction.xErr:=TRUE;
			T_Visu.T_CtrleAction.udiErrorID:=16#F1000 + T_Profile.T_Ctrle.iFunction;
			xAction_LoadProfileToProcessImage:=FALSE;
		END_CASE
	END_IF

(* Save profile to File *)
	IF xAction_SaveProfileToFile THEN
				(* Step import/export profile value *)
		CASE iStepAction OF
		(* Display message to ask for confirmation *)
		1:	IF T_Visu.ptrT_ExchgParam^.T_ProfileCommon.T_Id.iNumber > 1 THEN
				IF T_Visu.ptrT_ExchgParam^.T_ProfileCommon.T_Id.sName <> '' THEN
					IF NOT xFctCtrleProfileName(	sNewProfileName:=T_Visu.ptrT_ExchgParam^.T_ProfileCommon.T_Id.sName,
												ptrProfileList:=ADR(T_NovRam.T_Data.T_IDProfileStation)) THEN
						(* Display message 'ask for rewriting' *)
						T_Visu.ptrT_ExchgParam^.T_Visu.T_Message.iState:=112;
						(* next step *)
						iStepAction:=10;
					ELSE
						(* Display message 'confirm saving' *)
						T_Visu.ptrT_ExchgParam^.T_Visu.T_Message.iState:=108;
						(* next step *)
						iStepAction:=20;
					END_IF
				(* Display message, 'Profile name not correct' *)
				ELSE	tTimeOutAction:=TimerAction.ET+T#2s;
						T_Visu.ptrT_ExchgParam^.T_Visu.T_Message.iState:=16;
						iStepAction:=89;
				END_IF
			ELSE
				 tTimeOutAction:=TimerAction.ET+T#2s;
				T_Visu.ptrT_ExchgParam^.T_Visu.T_Message.iState:=6;
				iStepAction:=89;
			END_IF
		(* waiting for rewriting confirmation key <Enter> or <Esc> *)
		10:	IF RisingEdgeKeyPanel_Enter.Q THEN
			(* Display message *)
				T_Visu.ptrT_ExchgParam^.T_Visu.T_Message.iState:=13;
				(* next step *)
				iStepAction:=30;
			ELSE
				IF RisingEdgeKeyPanel_Esc.Q THEN iStepAction:=90; END_IF
				(* An other message has been displayed, stop saving action *)
				IF T_Visu.ptrT_ExchgParam^.T_Visu.T_Message.iState<>112 THEN iStepAction:=90; END_IF
			END_IF
		(* waiting for key <Enter> or <Esc> *)
		20:	IF RisingEdgeKeyPanel_Enter.Q THEN
			(* Display message *)
				T_Visu.ptrT_ExchgParam^.T_Visu.T_Message.iState:=13;
				(* next step *)
				iStepAction:=30;
			ELSE
				IF RisingEdgeKeyPanel_Esc.Q THEN iStepAction:=90; END_IF
				(* An other message has been displayed, stop saving action *)
				IF T_Visu.ptrT_ExchgParam^.T_Visu.T_Message.iState<>108 THEN iStepAction:=90; END_IF
			END_IF
		30:	(* page profile *)
			iTmp:=0;
			iTmp:=  iFctExistProfileName(	sProfileName:=T_Visu.ptrT_ExchgParam^.T_ProfileCommon.T_Id.sName,
										ptrProfileList:=ADR(T_NovRam.T_Data.T_IDProfileStation));
			IF iTmp = T_Visu.ptrT_ExchgParam^.T_ProfileCommon.T_Id.iNumber OR iTmp = 0 THEN
				IF NOT xFctCtrleProfileName(	sNewProfileName:=T_Visu.ptrT_ExchgParam^.T_ProfileCommon.T_Id.sName,
											ptrProfileList:=ADR(T_NovRam.T_Data.T_IDProfileStation)) THEN
					(* Rename profile datei *)
					sTmp:='\Hard Disk\Machine450\Profile\';
					sTmp_2:=sTmp;
					(* old name *)
					sTmp:=CONCAT(sTmp,T_NovRam.T_Data.T_IDProfileStation[T_Visu.ptrT_ExchgParam^.T_ProfileCommon.T_Id.iNumber].sName);
					T_HDD.T_File.sOldPathAndFileName:=CONCAT(sTmp,'.txt');
					(* new name *)
					sTmp_2:=CONCAT(sTmp_2,T_Visu.ptrT_ExchgParam^.T_ProfileCommon.T_Id.sName);
					T_HDD.T_File.sPathAndFileName:=CONCAT(sTmp_2,'.txt');
					IF T_HDD.T_File.sPathAndFileName<>T_HDD.T_File.sOldPathAndFileName THEN
					(* activ rename file *)
						T_HDD.T_Ctrle.xExecute:=TRUE;
						T_HDD.T_Ctrle.iFunction:=6;
					END_IF
				END_IF
				(* Disable Import prozess data state *)
				T_Visu.ptrT_ExchgParam^.T_ProfileCommon.xImportProzessData:=FALSE;
				(* next step *)
				iStepAction:=40;
			ELSE
				 tTimeOutAction:=TimerAction.ET+T#2s;
				T_Visu.ptrT_ExchgParam^.T_Visu.T_Message.iState:=24;
				iStepAction:=89;
			END_IF
		(* activ saving profile file *)
		40:	IF NOT T_HDD.T_Ctrle.xExecute AND T_HDD.T_Ctrle.xDone THEN
			(* activ saving profile file *)
				T_Profile.T_Id:=T_Visu.ptrT_ExchgParam^.T_ProfileCommon.T_Id;
				T_Profile.T_Ctrle.xExecute:=TRUE;
				T_Profile.T_Ctrle.iFunction:=2;
				(* next step *)
				iStepAction:=50;
			END_IF
			IF T_HDD.T_Ctrle.xErr THEN iStepAction:=99; END_IF
		(* waiting signal and start saving data in NovRAM *)
		50:	IF NOT T_Profile.T_Ctrle.xExecute AND T_Profile.T_Ctrle.xDone THEN
				T_NovRam.T_Data.T_IDProfileStation[T_Visu.ptrT_ExchgParam^.T_ProfileCommon.T_Id.iNumber]:=T_Visu.ptrT_ExchgParam^.T_ProfileCommon.T_Id;
(*				T_Visu.ptrT_ExchgParam^.T_StationCommon.T_InfoProcess.sProfileName  :=T_Visu.ptrT_ExchgParam^.T_ProfileCommon.T_Id.sName;      ausdokumentiert durch: unbekannt              *)
				(* Process profile value = file profile value *)
				IF T_Visu.ptrT_ExchgParam^.T_ProfileCommon.T_Id.iNumber = T_Visu.ptrT_ExchgParam^.T_StationCommon.T_InfoProcess.iProfile THEN
					T_NovRam.T_Data.T_ProcessImageLoadData:=T_NovRam.T_Data.T_ProcessImageData;
				END_IF
				(* page profile, update profile list *)
				xUpdateProfileList:=TRUE;
				(* next step *)
				iStepAction:=60;
			END_IF
			IF T_Profile.T_Ctrle.xErr THEN iStepAction:=99; END_IF

		(* active saving data NovRAM *)
		60:	xAction_SaveNovRAMWithoutConfirm:=TRUE;
			iStepActionNovRam:=1;
			(* next step *)
			iStepAction:=70;
		(* waiting confirm saving NovRAM action *)
		70:	IF NOT xAction_SaveNovRAMWithoutConfirm THEN
				iStepAction:=90;
			END_IF;
		(* no code, waiting timeout *)
		89:	IF TimerAction.Q THEN iStepAction:=90; END_IF
		(* save done *)
		90:	T_Visu.ptrT_ExchgParam^.T_Visu.T_Message.iState:=0;
			T_Visu.T_CtrleAction.xDone:=TRUE;
			T_Visu.T_CtrleAction.xNotReady:=FALSE;
			T_Visu.T_CtrleAction.xErr:=FALSE;
			T_Visu.T_CtrleAction.udiErrorID:=0;
			xAction_SaveProfileToFile:=FALSE;
		(* NovRAM not ready *)
		95:	TimerNotReady(IN:=TRUE);
			xAction_SaveProfileToFile:=FALSE;
		(* error *)
		99:	T_Visu.T_CtrleAction.xDone:=FALSE;
			T_Visu.T_CtrleAction.xNotReady:=FALSE;
			T_Visu.T_CtrleAction.xErr:=TRUE;
			T_Visu.T_CtrleAction.udiErrorID:=16#F0000 + T_Visu.T_CtrleAction.iFunction;
			IF T_HDD.T_Ctrle.xErr THEN T_Visu.T_CtrleAction.udiErrorID:=16#F1000 + T_HDD.T_Ctrle.iFunction; T_HDD.T_Ctrle.xReset:=TRUE; END_IF
			IF T_Profile.T_Ctrle.xErr THEN T_Visu.T_CtrleAction.udiErrorID:=16#F1000 + T_Visu.T_CtrleAction.iFunction; T_Profile.T_Ctrle.xReset:=TRUE; END_IF
			xAction_SaveProfileToFile:=FALSE;
		END_CASE
	END_IF;
(*SOA 27.01.2023    }   *)


(* Delete Profile *)
	IF xActionDeleteProfile THEN
		(* Step delete profile *)
		CASE iStepAction OF
		(* Profile number could not be 1 *)
		1:	IF T_Visu.ptrT_ExchgParam^.T_ProfileCommon.T_Id.iNumber < 2 THEN
				 tTimeOutAction:=TimerAction.ET+T#2s;
				T_Visu.ptrT_ExchgParam^.T_Visu.T_Message.iState:=27;	(* Default profile can't be deleted *)
				iStepAction:=10;
			ELSIF T_Visu.ptrT_ExchgParam^.T_StationCommon.T_InfoProcess.iProfile = T_Visu.ptrT_ExchgParam^.T_ProfileCommon.T_Id.iNumber THEN
				tTimeOutAction:=TimerAction.ET+T#2s;
				T_Visu.ptrT_ExchgParam^.T_Visu.T_Message.iState:=28;	(* Load profile can't be deleted *)
				iStepAction:=10;
			ELSE iStepAction:=20; END_IF
		(* no code, waiting timeout *)
		10:	IF TimerAction.Q THEN xActionDeleteProfile:=FALSE; END_IF;
		(* Display message to ask for confirmation *)
		20:	T_Visu.ptrT_ExchgParam^.T_Visu.T_Message.iState:=117;	(* Confirm delete profile <Enter>, or escape <Esc> ? *)
			(* next step *)
			iStepAction:=30;
		(* waiting for key <Enter> or <Esc> *)
		30:	IF RisingEdgeKeyPanel_Enter.Q THEN
				(* Display message deleting *)
				T_Visu.ptrT_ExchgParam^.T_Visu.T_Message.iState:=29;	(* Start deleting *)
				(* next step *)
				iStepAction:=40;
			ELSE
				IF RisingEdgeKeyPanel_Esc.Q THEN iStepAction:=90; END_IF
				(* An other message has been displayed, stop import/export action *)
				IF T_Visu.ptrT_ExchgParam^.T_Visu.T_Message.iState<>117 THEN iStepAction:=90; END_IF
			END_IF;
		(* Init. deleting profile file *)
		40:	IF T_NovRam.T_Data.T_IDProfileStation[T_Visu.ptrT_ExchgParam^.T_ProfileCommon.T_Id.iNumber].sName <> '' THEN
				sTmp:='\Hard Disk\Machine450\Profile\';
				sTmp:=CONCAT(sTmp,T_NovRam.T_Data.T_IDProfileStation[T_Visu.ptrT_ExchgParam^.T_ProfileCommon.T_Id.iNumber].sName);
				T_HDD.T_File.sPathAndFileName:=CONCAT(sTmp,'.txt');
				(* activ delete file *)
				T_HDD.T_Ctrle.xExecute:=TRUE;
				T_HDD.T_Ctrle.iFunction:=5;
				iStepAction:=50;
			(* Display info message 'file does not exists *)
			ELSE
				T_Visu.ptrT_ExchgParam^.T_Visu.T_Message.iState:=11;
				(* next step *)
				iStepAction:=55;
				xStepActionDone:=FALSE;
				tTimeOutAction:=TimerAction.ET+T#2s;
			END_IF
		50:	IF NOT T_HDD.T_Ctrle.xExecute AND (T_HDD.T_Ctrle.xDone OR T_HDD.T_Ctrle.xErr) THEN
				T_HDD.T_Ctrle.xReset:=T_HDD.T_Ctrle.xErr;
				(* Profile will be erased from the profile list *)
				T_NovRam.T_Data.T_IDProfileStation[T_Visu.ptrT_ExchgParam^.T_ProfileCommon.T_Id.iNumber].sName:='';
				xUpdateProfileList:=TRUE;
				IF T_HDD.T_Ctrle.xErr THEN
					(* Display info message 'file does not exists *)
					T_Visu.ptrT_ExchgParam^.T_Visu.T_Message.iState:=11;
					(* next step *)
					iStepAction:=52;
					xStepActionDone:=FALSE;
					(* use tmp timer to diplay message *)
					TimerONTmp(IN:=FALSE);
					TimerONTmp.PT:=T#2s;
				ELSE
					(* next step *)
					iStepAction:=70;
					xStepActionDone:=FALSE;
				END_IF;
			END_IF
		(* Wait delay timer *)
		52:	IF TimerONTmp.Q THEN
				T_Visu.ptrT_ExchgParam^.T_Visu.T_Message.iState:=0;
				(* next step *)
				iStepAction:=70;
			END_IF
		(* delay time out *)
		55:	IF TimerAction.Q THEN xActionDeleteProfile:=FALSE; END_IF
		(* active saving data NovRAM *)
		70:	T_Visu.ptrT_ExchgParam^.T_ProfileCommon.T_Id.sName:='';
			xAction_SaveNovRAMWithoutConfirm:=TRUE;
			iStepActionNovRam:=1;
			(* next step *)
			iStepAction:=80;
		(* waiting confirm saving NovRAM action *)
		80:	IF NOT xAction_SaveNovRAMWithoutConfirm THEN iStepAction:=90; END_IF
		(* save done *)
		90:	T_Visu.ptrT_ExchgParam^.T_Visu.T_Message.iState:=0;
			T_Visu.T_CtrleAction.xDone:=TRUE;
			T_Visu.T_CtrleAction.xNotReady:=FALSE;
			T_Visu.T_CtrleAction.xErr:=FALSE;
			T_Visu.T_CtrleAction.udiErrorID:=0;
			xActionDeleteProfile:=FALSE;
		(* Action not ready *)
		95:	TimerNotReady(IN:=TRUE);
			xActionDeleteProfile:=FALSE;
		(* error *)
		99:	T_Visu.T_CtrleAction.xDone:=FALSE;
			T_Visu.T_CtrleAction.xNotReady:=FALSE;
			T_Visu.T_CtrleAction.xErr:=TRUE;
			T_Visu.T_CtrleAction.udiErrorID:=16#F1000 + T_Profile.T_Ctrle.iFunction;
			xActionDeleteProfile:=FALSE;
		END_CASE;
	END_IF;
END_ACTION
ACTION VisuFunction_SetParameterPage:
(* Action set parameter page *)
	IF xSetParameterPage THEN
		(* set parameter page *)
		CASE iStepAction OF
		(* check visu *)
		1:	IF (T_Visu.T_PlcParam.dwActualPage = 140) OR (T_Visu.T_PlcParam.dwActualPage = 150) THEN
				(* For this page. for select the parameter list, it need the system level *)
				IF (T_ExchgParam.T_Visu.T_Level.iActLevel <> 2) THEN
					T_ExchgParam.T_Visu.T_Message.iState:=36;	(* Display Message --> This parameter can be change only with system level *)
						T_Visu.ptrT_ExchgParam^.T_TouchScreenBtPanel.iStateBtLeft:=WORD_TO_INT(INT_TO_WORD(T_Visu.ptrT_ExchgParam^.T_TouchScreenBtPanel.iStateBtLeft) AND 16#FFEF);
				END_IF;
			END_IF;
			IF (T_ExchgParam.T_Visu.T_Message.iState <> 36) THEN
				xTmp:=	T_Visu.T_CtrleVisu.xDone
						AND NOT(T_Visu.T_CtrleVisu.xExecute)
						AND NOT(T_Visu.T_CtrleVisu.xErr);
				IF xTmp THEN
					(* next Step *)
					iStepAction :=10;
					xStepActionDone:=FALSE;
				(* activ error *)
				ELSE iStepAction:=95; END_IF
			ELSE
				iStepAction:=90;
			END_IF;
		(* Set parameter page *)
		10:	T_Visu.ptrT_ExchgParam^.T_Config.xBlockParaListNavi:=FALSE;
			T_Visu.ptrT_ExchgParam^.T_Config.xBlockParaListNavi1:=TRUE;
			T_Visu.ptrT_ExchgParam^.T_Config.xBlockProfilList:=TRUE;
			CASE T_Visu.ptrT_ExchgParam^.T_Visu.bActivSpecialLayer OF
				1:	T_Visu.T_PlcParam.dwSetNewPage:=170;
					T_Visu.ptrT_ExchgParam^.T_Config.iEditParam:=iFctGetEditParaList(	dwActualPage:=wSpecialLayerGeneralActivPage,
																				xMicroRodActive:=xMicroRodActive,
																				iSelectParaList:=T_Visu.ptrT_ExchgParam^.T_Config.iSelectParaList,
																				iSelectParaListTeachRot:=T_Visu.ptrT_ExchgParam^.T_Config.iSelectParaListTeachRot);
					IF (T_Visu.ptrT_ExchgParam^.T_Config.iEditParam = 140) OR (T_Visu.ptrT_ExchgParam^.T_Config.iEditParam = 150) THEN
						(* For this page. for select the parameter list, it need the system level *)
						IF (T_ExchgParam.T_Visu.T_Level.iActLevel <> 2) THEN
							T_ExchgParam.T_Visu.T_Message.iState:=36;	(* Display Message --> This parameter can be change only with system level *)
								T_Visu.ptrT_ExchgParam^.T_TouchScreenBtPanel.iStateBtLeft:=WORD_TO_INT(INT_TO_WORD(T_Visu.ptrT_ExchgParam^.T_TouchScreenBtPanel.iStateBtLeft) AND 16#FFEF);
								T_Visu.T_PlcParam.dwSetNewPage:=wSpecialLayerGeneralActivPage;
						END_IF;
					END_IF;
					IF (T_ExchgParam.T_Visu.T_Message.iState <> 36) THEN
						(* 09.12.2010 KFS:	{	*)
						IF (T_ExchgParam.T_Visu.T_Level.iActLevel =2) THEN
						(* 09.12.2010 KFS:	}	*)
							IF (T_Visu.ptrT_ExchgParam^.T_Config.iEditParam = 110) OR (T_Visu.ptrT_ExchgParam^.T_Config.iEditParam = 111) THEN
								T_Visu.ptrT_ExchgParam^.T_Config.xBlockProfilList:=FALSE;
							END_IF;
							IF ((T_Visu.ptrT_ExchgParam^.T_Config.iEditParam >= 120) AND (T_Visu.ptrT_ExchgParam^.T_Config.iEditParam <= 129)) THEN
								T_Visu.ptrT_ExchgParam^.T_Config.xBlockProfilList:=FALSE;
							END_IF;
							IF (T_Visu.ptrT_ExchgParam^.T_Config.iEditParam = 130) OR (T_Visu.ptrT_ExchgParam^.T_Config.iEditParam = 131) THEN
								T_Visu.ptrT_ExchgParam^.T_Config.xBlockParaListNavi1:=FALSE;
								T_Visu.ptrT_ExchgParam^.T_Config.xBlockParaListNavi:=TRUE;
								T_Visu.ptrT_ExchgParam^.T_Config.xBlockProfilList:=FALSE;
								(*  Set Loaded Profil Data from the read file*)
								T_Visu.ptrT_ExchgParam^.T_StationCommon.T_AutoGeometryPara:=T_NovRAM.T_Data.T_ProcessImageLoadData.T_AutoGeometryPara;
								T_Visu.ptrT_ExchgParam^.T_StationCommon.T_AutoGroovePara:=T_NovRAM.T_Data.T_ProcessImageLoadData.T_AutoGroovePara;
								T_Visu.ptrT_ExchgParam^.T_StationCommon.T_CalibrationPara:=T_NovRAM.T_Data.T_ProcessImageLoadData.T_CalibrationPara;
								T_Visu.ptrT_ExchgParam^.T_StationCommon.T_ProcessPara:=T_NovRAM.T_Data.T_ProcessImageLoadData.T_ProcessPara;
								T_Visu.ptrT_ExchgParam^.T_GeometryCommon.T_Geometry:=T_NovRAM.T_Data.T_ProcessImageLoadData.T_GeometryPara;
								T_Visu.ptrT_ExchgParam^.T_StationCommon.T_PrismPara:=T_NovRAM.T_Data.T_ProcessImageLoadData.T_PrismPara;
							END_IF;
							IF (T_Visu.ptrT_ExchgParam^.T_Config.iEditParam = 150) THEN
								T_Visu.ptrT_ExchgParam^.T_Config.xBlockParaListNavi:=TRUE;
							END_IF;
						(* 09.12.2010 KFS:	{	*)
						ELSE
							IF (T_Visu.ptrT_ExchgParam^.T_Config.iEditParam = 110) OR (T_Visu.ptrT_ExchgParam^.T_Config.iEditParam = 111) THEN
								IF  (T_Visu.ptrT_ExchgParam^.T_Config.iEditParam = 111) THEN
									 T_Visu.ptrT_ExchgParam^.T_Config.iEditParam:= 112;
								END_IF;
								T_Visu.ptrT_ExchgParam^.T_Config.xBlockProfilList:=FALSE;
							END_IF;
							IF ((T_Visu.ptrT_ExchgParam^.T_Config.iEditParam >= 120) AND (T_Visu.ptrT_ExchgParam^.T_Config.iEditParam <= 129)) THEN
								IF  (T_Visu.ptrT_ExchgParam^.T_Config.iEditParam = 121) THEN
									 T_Visu.ptrT_ExchgParam^.T_Config.iEditParam:= 126;
								ELSIF ( T_Visu.ptrT_ExchgParam^.T_Config.iEditParam = 123) THEN
									 T_Visu.ptrT_ExchgParam^.T_Config.iEditParam:= 127;
								ELSIF ( T_Visu.ptrT_ExchgParam^.T_Config.iEditParam = 125) THEN
									 T_Visu.ptrT_ExchgParam^.T_Config.iEditParam:= 128;
								END_IF;
								T_Visu.ptrT_ExchgParam^.T_Config.xBlockProfilList:=FALSE;
							END_IF;
							IF (T_Visu.ptrT_ExchgParam^.T_Config.iEditParam = 130) OR (T_Visu.ptrT_ExchgParam^.T_Config.iEditParam = 131) THEN
								T_Visu.ptrT_ExchgParam^.T_Config.xBlockParaListNavi1:=FALSE;
								T_Visu.ptrT_ExchgParam^.T_Config.xBlockParaListNavi:=TRUE;
								T_Visu.ptrT_ExchgParam^.T_Config.xBlockProfilList:=FALSE;
								(*  Set Loaded Profil Data from the read file*)
								T_Visu.ptrT_ExchgParam^.T_StationCommon.T_AutoGeometryPara:=T_NovRAM.T_Data.T_ProcessImageLoadData.T_AutoGeometryPara;
								T_Visu.ptrT_ExchgParam^.T_StationCommon.T_AutoGroovePara:=T_NovRAM.T_Data.T_ProcessImageLoadData.T_AutoGroovePara;
								T_Visu.ptrT_ExchgParam^.T_StationCommon.T_CalibrationPara:=T_NovRAM.T_Data.T_ProcessImageLoadData.T_CalibrationPara;
								T_Visu.ptrT_ExchgParam^.T_StationCommon.T_ProcessPara:=T_NovRAM.T_Data.T_ProcessImageLoadData.T_ProcessPara;
								T_Visu.ptrT_ExchgParam^.T_GeometryCommon.T_Geometry:=T_NovRAM.T_Data.T_ProcessImageLoadData.T_GeometryPara;
								T_Visu.ptrT_ExchgParam^.T_StationCommon.T_PrismPara:=T_NovRAM.T_Data.T_ProcessImageLoadData.T_PrismPara;
							END_IF;
							IF (T_Visu.ptrT_ExchgParam^.T_Config.iEditParam = 150) THEN
								T_Visu.ptrT_ExchgParam^.T_Config.xBlockParaListNavi:=TRUE;
							END_IF;
						END_IF;
						(* 09.12.2010 KFS:	}	*)
					END_IF;
				2:	T_Visu.T_PlcParam.dwSetNewPage:=270;
					T_Visu.ptrT_ExchgParam^.T_Config.iEditParam:=iFctGetEditParaList(	dwActualPage:=wSpecialLayerToolRotActivPage,
																				xMicroRodActive:=xMicroRodActive,
																				iSelectParaList:=T_Visu.ptrT_ExchgParam^.T_Config.iSelectParaList,
																				iSelectParaListTeachRot:=T_Visu.ptrT_ExchgParam^.T_Config.iSelectParaListTeachRot);
				3:	T_Visu.T_PlcParam.dwSetNewPage:=370;
					T_Visu.ptrT_ExchgParam^.T_Config.iEditParam:=iFctGetEditParaList(	dwActualPage:=wSpecialLayerWireFeedActivPage,
																				xMicroRodActive:=xMicroRodActive,
																				iSelectParaList:=T_Visu.ptrT_ExchgParam^.T_Config.iSelectParaList,
																				iSelectParaListTeachRot:=T_Visu.ptrT_ExchgParam^.T_Config.iSelectParaListTeachRot);
				4:	T_Visu.T_PlcParam.dwSetNewPage:=470;
					T_Visu.ptrT_ExchgParam^.T_Config.iEditParam:=iFctGetEditParaList(	dwActualPage:=wSpecialLayerGrindAxisActivPage,
																				xMicroRodActive:=xMicroRodActive,
																				iSelectParaList:=T_Visu.ptrT_ExchgParam^.T_Config.iSelectParaList,
																				iSelectParaListTeachRot:=T_Visu.ptrT_ExchgParam^.T_Config.iSelectParaListTeachRot);
			END_CASE;
			T_Visu.T_CtrleVisu.iFunction:=1;
			T_Visu.T_CtrleVisu.xExecute:=TRUE;
			(* activ step *)
			iStepAction:=20;
			xStepActionDone:=FALSE;
		(* wait for changing page *)
		20:	IF NOT(xStepActionDone) THEN
			(* release execution *)
				T_Visu.T_CtrleVisu.xExecute:=FALSE;
				(* confirm step done *)
				xStepActionDone:=TRUE;
			ELSE
				IF T_Visu.T_CtrleVisu.xDone THEN
				(* activ next step *)
					iStepAction:=90;
					xStepActionDone:=FALSE;
				END_IF
				IF T_Visu.T_CtrleVisu.xErr THEN
				(* activ next error *)
					iStepAction:=99;
					xStepActionDone:=FALSE;
				END_IF
			END_IF
		(* change page done *)
		90:	T_Visu.T_CtrleAction.xDone:=TRUE;
			T_Visu.T_CtrleAction.xNotReady:=FALSE;
			T_Visu.T_CtrleAction.xErr:=FALSE;
			T_Visu.T_CtrleAction.udiErrorID:=0;
			xSetParameterPage:=FALSE;
		(* override done *)
		91:	T_Visu.T_CtrleAction.xDone:=TRUE;
			T_Visu.T_CtrleAction.xNotReady:=FALSE;
			T_Visu.T_CtrleAction.xErr:=FALSE;
			T_Visu.T_CtrleAction.udiErrorID:=0;
			xSetParameterPage:=FALSE;
		(* not ready *)
		95:	T_Visu.T_CtrleAction.xDone:=TRUE;
			T_Visu.T_CtrleAction.xNotReady:=FALSE;
			T_Visu.T_CtrleAction.xErr:=FALSE;
			T_Visu.T_CtrleAction.udiErrorID:=0;
			xSetParameterPage:=FALSE;
		(* error *)
		99:	T_Visu.T_CtrleAction.xDone:=FALSE;
			T_Visu.T_CtrleAction.xNotReady:=FALSE;
			T_Visu.T_CtrleAction.xErr:=TRUE;
			T_Visu.T_CtrleAction.udiErrorID:=16#F0000 + T_Visu.T_CtrleAction.iFunction;
			xSetParameterPage:=FALSE;
		END_CASE
	END_IF
END_ACTION
ACTION VisuFunction_SetupSection:
(* Activation of the Section for the ToolGeometry *)
	IF xActivationSection1 OR xActivationSection2 OR xActivationSection3 OR xActivationSection4 OR xActivationSection5 OR xActivationSection6 OR xSetPitchEqual THEN
		CASE iStepAction OF
		(* check visu *)
		1:	xTmp:=	TRUE;
			IF xTmp THEN
				(* next Step *)
				iStepAction :=10;
			(* activ error *)
			ELSE iStepAction:=95; END_IF
		(* Set parameter page *)
		10:	ptxActiveSection1:=ADR(T_Visu.ptrT_ExchgParam^.T_GeometryCommon.T_Geometry.axActiveSection[1]);
			ptxActiveSection2:=ADR(T_Visu.ptrT_ExchgParam^.T_GeometryCommon.T_Geometry.axActiveSection[2]);
			ptxActiveSection3:=ADR(T_Visu.ptrT_ExchgParam^.T_GeometryCommon.T_Geometry.axActiveSection[3]);
			ptxActiveSection4:=ADR(T_Visu.ptrT_ExchgParam^.T_GeometryCommon.T_Geometry.axActiveSection[4]);
			ptxActiveSection5:=ADR(T_Visu.ptrT_ExchgParam^.T_GeometryCommon.T_Geometry.axActiveSection[5]);
			ptxActiveSection6:=ADR(T_Visu.ptrT_ExchgParam^.T_GeometryCommon.T_Geometry.axActiveSection[6]);

(*** Checking if: the section is already active / is the olny active / a section before is active  ***)
			IF xActivationSection1 THEN
				IF (ptxActiveSection1^ AND NOT(ptxActiveSection2^)) OR
				     (NOT(ptxActiveSection1^) AND NOT(ptxActiveSection2^) AND (ptxActiveSection3^ OR ptxActiveSection4^OR ptxActiveSection5^ OR ptxActiveSection6^)) THEN
					;
				ELSE
					ptxActiveSection1^:=NOT(ptxActiveSection1^);
				END_IF;
			END_IF;

			IF xActivationSection2 THEN
				IF (ptxActiveSection2^ AND ptxActiveSection1^ AND ptxActiveSection3^) OR
				    (ptxActiveSection2^ AND NOT(ptxActiveSection1^) AND NOT(ptxActiveSection3^)) OR
				    (NOT(ptxActiveSection2^) AND NOT(ptxActiveSection1^) AND NOT(ptxActiveSection3^) AND (ptxActiveSection4^OR ptxActiveSection5^ OR ptxActiveSection6^)) THEN
					;
				ELSE
					ptxActiveSection2^:=NOT(ptxActiveSection2^);
				END_IF;
			END_IF;
				IF xActivationSection3 THEN
					IF (ptxActiveSection3^ AND ptxActiveSection2^ AND ptxActiveSection4^) OR
					    (ptxActiveSection3^ AND NOT(ptxActiveSection2^) AND NOT(ptxActiveSection4^)) OR
					    (NOT(ptxActiveSection3^) AND NOT(ptxActiveSection2^) AND NOT(ptxActiveSection4^) AND (ptxActiveSection5^ OR ptxActiveSection6^ OR ptxActiveSection1^))THEN
						;
					ELSE
						ptxActiveSection3^:=NOT(ptxActiveSection3^);
					END_IF;
				END_IF;
			IF xActivationSection4 THEN
				IF (ptxActiveSection4^ AND ptxActiveSection3^ AND ptxActiveSection5^) OR
				    (ptxActiveSection4^ AND NOT(ptxActiveSection3^) AND NOT(ptxActiveSection5^)) OR
				    (NOT(ptxActiveSection4^) AND NOT(ptxActiveSection3^) AND NOT(ptxActiveSection5^) AND (ptxActiveSection6^OR ptxActiveSection1^ OR ptxActiveSection2^)) THEN
					;
				ELSE
					ptxActiveSection4^:=NOT(ptxActiveSection4^);
				END_IF;
			END_IF;
(*09.12.2022: SOA	{	 *)
				IF xActivationSection5 THEN
					IF (ptxActiveSection5^ AND ptxActiveSection4^ AND ptxActiveSection6^) OR
					    (ptxActiveSection5^ AND NOT(ptxActiveSection4^) AND NOT(ptxActiveSection6^)) OR
					    (NOT(ptxActiveSection5^) AND NOT(ptxActiveSection4^) AND NOT(ptxActiveSection6^) AND (ptxActiveSection1^ OR ptxActiveSection2^ OR ptxActiveSection3^))THEN
						;
					ELSE
						ptxActiveSection5^:=NOT(ptxActiveSection5^);
					END_IF;
				END_IF;
			IF xActivationSection6 THEN
				IF (ptxActiveSection6^ AND NOT(ptxActiveSection5^)) OR
				    (NOT(ptxActiveSection6^) AND NOT(ptxActiveSection5^) AND (ptxActiveSection1^ OR ptxActiveSection2^ OR ptxActiveSection3^ OR ptxActiveSection4^ )) THEN
					;
				ELSE
					ptxActiveSection6^:=NOT(ptxActiveSection6^);
				END_IF;
			END_IF;
(*09.12.2022: SOA	}	 *)
(*09.12.2022: SOA	{	 *)
			IF xSetPitchEqual THEN
				IF T_Visu.ptrT_ExchgParam^.T_GeometryCommon.T_Geometry.axActiveSection[1] THEN
					rSectionPitch:=T_Visu.ptrT_ExchgParam^.T_GeometryCommon.T_Geometry.arSectionPitch[1];
					IF T_Visu.ptrT_ExchgParam^.T_GeometryCommon.T_Geometry.axActiveSection[2] THEN
						T_Visu.ptrT_ExchgParam^.T_GeometryCommon.T_Geometry.arSectionPitch[2]:=rSectionPitch;
					END_IF;
					IF T_Visu.ptrT_ExchgParam^.T_GeometryCommon.T_Geometry.axActiveSection[3] THEN
						T_Visu.ptrT_ExchgParam^.T_GeometryCommon.T_Geometry.arSectionPitch[3]:=rSectionPitch;
					END_IF;
					IF T_Visu.ptrT_ExchgParam^.T_GeometryCommon.T_Geometry.axActiveSection[4] THEN
						T_Visu.ptrT_ExchgParam^.T_GeometryCommon.T_Geometry.arSectionPitch[4]:=rSectionPitch;
					END_IF;
					IF T_Visu.ptrT_ExchgParam^.T_GeometryCommon.T_Geometry.axActiveSection[5] THEN
						T_Visu.ptrT_ExchgParam^.T_GeometryCommon.T_Geometry.arSectionPitch[5]:=rSectionPitch;
					END_IF;
					IF T_Visu.ptrT_ExchgParam^.T_GeometryCommon.T_Geometry.axActiveSection[6] THEN
						T_Visu.ptrT_ExchgParam^.T_GeometryCommon.T_Geometry.arSectionPitch[6]:=rSectionPitch;
					END_IF;
				ELSIF T_Visu.ptrT_ExchgParam^.T_GeometryCommon.T_Geometry.axActiveSection[2] THEN
					rSectionPitch:=T_Visu.ptrT_ExchgParam^.T_GeometryCommon.T_Geometry.arSectionPitch[2];
					IF T_Visu.ptrT_ExchgParam^.T_GeometryCommon.T_Geometry.axActiveSection[3] THEN
						T_Visu.ptrT_ExchgParam^.T_GeometryCommon.T_Geometry.arSectionPitch[3]:=rSectionPitch;
					END_IF;
					IF T_Visu.ptrT_ExchgParam^.T_GeometryCommon.T_Geometry.axActiveSection[4] THEN
						T_Visu.ptrT_ExchgParam^.T_GeometryCommon.T_Geometry.arSectionPitch[4]:=rSectionPitch;
					END_IF;
					IF T_Visu.ptrT_ExchgParam^.T_GeometryCommon.T_Geometry.axActiveSection[5] THEN
						T_Visu.ptrT_ExchgParam^.T_GeometryCommon.T_Geometry.arSectionPitch[5]:=rSectionPitch;
					END_IF;
					IF T_Visu.ptrT_ExchgParam^.T_GeometryCommon.T_Geometry.axActiveSection[6] THEN
						T_Visu.ptrT_ExchgParam^.T_GeometryCommon.T_Geometry.arSectionPitch[6]:=rSectionPitch;
					END_IF;
				ELSIF T_Visu.ptrT_ExchgParam^.T_GeometryCommon.T_Geometry.axActiveSection[3] THEN
					rSectionPitch:=T_Visu.ptrT_ExchgParam^.T_GeometryCommon.T_Geometry.arSectionPitch[3];
					IF T_Visu.ptrT_ExchgParam^.T_GeometryCommon.T_Geometry.axActiveSection[4] THEN
						T_Visu.ptrT_ExchgParam^.T_GeometryCommon.T_Geometry.arSectionPitch[4]:=rSectionPitch;
					END_IF;
					IF T_Visu.ptrT_ExchgParam^.T_GeometryCommon.T_Geometry.axActiveSection[5] THEN
						T_Visu.ptrT_ExchgParam^.T_GeometryCommon.T_Geometry.arSectionPitch[5]:=rSectionPitch;
					END_IF;
					IF T_Visu.ptrT_ExchgParam^.T_GeometryCommon.T_Geometry.axActiveSection[6] THEN
						T_Visu.ptrT_ExchgParam^.T_GeometryCommon.T_Geometry.arSectionPitch[6]:=rSectionPitch;
					END_IF;
				ELSIF T_Visu.ptrT_ExchgParam^.T_GeometryCommon.T_Geometry.axActiveSection[4] THEN
					rSectionPitch:=T_Visu.ptrT_ExchgParam^.T_GeometryCommon.T_Geometry.arSectionPitch[4];
					IF T_Visu.ptrT_ExchgParam^.T_GeometryCommon.T_Geometry.axActiveSection[5] THEN
						T_Visu.ptrT_ExchgParam^.T_GeometryCommon.T_Geometry.arSectionPitch[5]:=rSectionPitch;
					END_IF;
					IF T_Visu.ptrT_ExchgParam^.T_GeometryCommon.T_Geometry.axActiveSection[6] THEN
						T_Visu.ptrT_ExchgParam^.T_GeometryCommon.T_Geometry.arSectionPitch[6]:=rSectionPitch;
					END_IF;
				ELSIF T_Visu.ptrT_ExchgParam^.T_GeometryCommon.T_Geometry.axActiveSection[5] THEN
					rSectionPitch:=T_Visu.ptrT_ExchgParam^.T_GeometryCommon.T_Geometry.arSectionPitch[5];
					IF T_Visu.ptrT_ExchgParam^.T_GeometryCommon.T_Geometry.axActiveSection[6] THEN
						T_Visu.ptrT_ExchgParam^.T_GeometryCommon.T_Geometry.arSectionPitch[6]:=rSectionPitch;
					END_IF;
				ELSIF T_Visu.ptrT_ExchgParam^.T_GeometryCommon.T_Geometry.axActiveSection[6] THEN
					rSectionPitch:=T_Visu.ptrT_ExchgParam^.T_GeometryCommon.T_Geometry.arSectionPitch[6];
				END_IF;
			END_IF;
(*09.12.2022: SOA	}   *)
			iStepAction :=90;
		(* change page done *)
		90:	T_Visu.T_CtrleAction.xDone:=TRUE;
			T_Visu.T_CtrleAction.xNotReady:=FALSE;
			T_Visu.T_CtrleAction.xErr:=FALSE;
			T_Visu.T_CtrleAction.udiErrorID:=0;
			xActivationSection1:=xActivationSection2:=xActivationSection3:=xActivationSection4:=xActivationSection5:=xActivationSection6:=xSetPitchEqual:=FALSE;
		(* not ready *)
		95:	T_Visu.T_CtrleAction.xDone:=TRUE;
			T_Visu.T_CtrleAction.xNotReady:=FALSE;
			T_Visu.T_CtrleAction.xErr:=FALSE;
			T_Visu.T_CtrleAction.udiErrorID:=0;
			xActivationSection1:=xActivationSection2:=xActivationSection3:=xActivationSection4:=xActivationSection5:=xActivationSection6:=xSetPitchEqual:=FALSE;
		(* error *)
		99:	T_Visu.T_CtrleAction.xDone:=FALSE;
			T_Visu.T_CtrleAction.xNotReady:=FALSE;
			T_Visu.T_CtrleAction.xErr:=TRUE;
			T_Visu.T_CtrleAction.udiErrorID:=16#F0000 + T_Visu.T_CtrleAction.iFunction;
			xActivationSection1:=xActivationSection2:=xActivationSection3:=xActivationSection4:=xActivationSection5:=xActivationSection6:=xSetPitchEqual:=FALSE;
		END_CASE
	END_IF;
END_ACTION
ACTION VisuFunction_SetupWarmup:
(************************************************************************************************************************************************************************)
(***************                                             start of warmup section 														     ********************)
(************************************************************************************************************************************************************************)

(* SOA 12.01.2023  {   *)
	(* Warmup Wochentage auswählen*)
	IF T_Visu.T_PlcParam.dwActualPage = 141 THEN
	(*	T_ExchgParam.T_FunctionCommon.xWarmUp_ContactorMachine_Active:= FALSE; (* xWarmUp;*) (*QxTwinSafe_Machine_ON;*) (*	xWarmUp := FALSE; *) ***Delete***   *)
		FOR ii:=0 TO 6 DO
			(* Wochentage auswählen *)
			IF T_ExchgParam.T_FunctionCommon.axWarmUp_DayOfWeekButton[ii] THEN
				T_ExchgParam.T_FunctionCommon.axWarmUp_DayOfWeekButton[ii]:=FALSE;
				T_ExchgParam.T_FunctionCommon.TWarmUp_Para.axDayOfWeek[ii]:=NOT(T_ExchgParam.T_FunctionCommon.TWarmUp_Para.axDayOfWeek[ii]);
				iCountDayOfWeek:=0;
				FOR jj:=0 TO 6 DO
					IF T_ExchgParam.T_FunctionCommon.TWarmUp_Para.axDayOfWeek[jj] THEN
						iCountDayOfWeek:=iCountDayOfWeek + 1;
					END_IF;
				END_FOR;
				IF (iCountDayOfWeek = 0) THEN
					T_ExchgParam.T_FunctionCommon.TWarmUp_Para.axDayOfWeek[ii]:=TRUE;	(* Darf nicht ausgeschaltet werden, da sonst kein Wochentag gesetzt ist *)
					T_ExchgParam.T_Visu.T_Message.iState:=51;	(* Warnung: Mindestens ein Wochentag muss gesetzt sein ! *)
				END_IF;
			END_IF;
		END_FOR;
		(* Wochentag überprüfen *)
		xReadyToCheckWarmUp:=FALSE;
		CASE T_ExchgParam.T_TimeStamp.wDayOfWeek OF
		(* Sonntag *)
		0:	IF T_ExchgParam.T_FunctionCommon.TWarmUp_Para.axDayOfWeek[0] THEN
				xReadyToCheckWarmUp:=TRUE;
			END_IF;
		(* Montag *)
		1:	IF T_ExchgParam.T_FunctionCommon.TWarmUp_Para.axDayOfWeek[1] THEN
				xReadyToCheckWarmUp:=TRUE;
			END_IF;
		(* Dienstag *)
		2:	IF T_ExchgParam.T_FunctionCommon.TWarmUp_Para.axDayOfWeek[2] THEN
				xReadyToCheckWarmUp:=TRUE;
			END_IF;
		(* Mittwoch *)
		3:	IF T_ExchgParam.T_FunctionCommon.TWarmUp_Para.axDayOfWeek[3] THEN
				xReadyToCheckWarmUp:=TRUE;
			END_IF;
		(* Donnerstag *)
		4:	IF T_ExchgParam.T_FunctionCommon.TWarmUp_Para.axDayOfWeek[4] THEN
				xReadyToCheckWarmUp:=TRUE;
			END_IF;
		(* Freitag *)
		5:	IF T_ExchgParam.T_FunctionCommon.TWarmUp_Para.axDayOfWeek[5] THEN
				xReadyToCheckWarmUp:=TRUE;
			END_IF;
		(* Samstag *)
		6:	IF T_ExchgParam.T_FunctionCommon.TWarmUp_Para.axDayOfWeek[6] THEN
				xReadyToCheckWarmUp:=TRUE;
			END_IF;
		END_CASE;

		wConvertMinute:=REAL_TO_WORD((WORD_TO_REAL(T_ExchgParam.T_TimeStamp.wMinute)/60.0) * 100.0);
		IF (wConvertMinute > 100) THEN wConvertMinute:=100; END_IF;
		wCheckTimeWarmUp:=(T_ExchgParam.T_TimeStamp.wHour * 100) + wConvertMinute;

		wConertMinute_StartTime:=REAL_TO_WORD((INT_TO_REAL(T_NovRam.T_Data.TWarmUp_Para.iWarmUp_TimeON_Minute)/60.0) * 100.0);
		IF (wConertMinute_StartTime > 100) THEN wConertMinute_StartTime:=100; END_IF;
		wCheckTimeWarmUp_StartTime:=(T_NovRam.T_Data.TWarmUp_Para.iWarmUp_TimeON_Hour * 100) + wConertMinute_StartTime;

		wConertMinute_StopTime:=REAL_TO_WORD((INT_TO_REAL(T_NovRam.T_Data.TWarmUp_Para.iWarmUp_TimeOFF_Minute)/60.0) * 100.0);
		IF (wConertMinute_StopTime > 100) THEN wConertMinute_StopTime:=100; END_IF;
		wCheckTimeWarmUp_StopTime:=(T_NovRam.T_Data.TWarmUp_Para.iWarmUp_TimeOFF_Hour * 100) + wConertMinute_StopTime;


		xReadyToStartNextTime:=xWarmuUp_Start:=xWarmUp_Stop:=FALSE;
		IF xReadyToCheckWarmUp THEN
			IF (wCheckTimeWarmUp >= (wCheckTimeWarmUp_StartTime - 2)) THEN
				xReadyToStartNextTime:=TRUE;
			END_IF;
			IF (wCheckTimeWarmUp >= wCheckTimeWarmUp_StartTime) THEN
				xWarmuUp_Start:=TRUE;
			END_IF;
			IF (wCheckTimeWarmUp >= wCheckTimeWarmUp_StopTime) THEN
				xWarmUp_Stop:=TRUE;
				xConfirmStartWarmUp:=FALSE;
			END_IF;
		END_IF;
		IF NOT (T_TwinSafeIn.IxContactorAuxContact) THEN (* IF NOT(T_TwinSafeIn.IxAxesCurrentOffCh1) AND NOT(T_TwinSafeIn.IxAxesCurrentOffCh2) THEN (****TODO****) *)   		(*Eventuell:	xContactor_K3:BOOL;	QxContactor_K4:BOOL;*)
			IF xWarmUp_Stop THEN
				T_ExchgParam.T_FunctionCommon.xWarmUp_ContactorMachine_Active:= FALSE;
			ELSIF xReadyToStartNextTime AND xWarmuUp_Start AND xStartUpConfirmed THEN
				T_ExchgParam.T_FunctionCommon.xWarmUp_ContactorMachine_Active:= TRUE;
				T_ExchgParam.T_FunctionCommon.xWarmUp_MessageWarning:=FALSE;
			ELSIF xReadyToStartNextTime AND xStartUpConfirmed THEN
				T_ExchgParam.T_FunctionCommon.xWarmUp_ContactorMachine_Active:= FALSE;
				T_ExchgParam.T_FunctionCommon.xWarmUp_MessageWarning:=TRUE;
			END_IF;
		ELSE
			T_ExchgParam.T_FunctionCommon.xWarmUp_ContactorMachine_Active:= FALSE;
			T_ExchgParam.T_FunctionCommon.xWarmUp_MessageWarning:=FALSE;
		END_IF;
		TONWarmUpChangeColour(IN:=TRUE,PT:=T#1s);
		IF TONWarmUpChangeColour.Q THEN
			TONWarmUpChangeColour(IN:=FALSE);
			IF T_ExchgParam.T_FunctionCommon.xWarmUp_MessageWarning THEN
				T_ExchgParam.T_FunctionCommon.iWarmUp_ColourChange:=T_ExchgParam.T_FunctionCommon.iWarmUp_ColourChange XOR 1;
			END_IF;
		END_IF;
	ELSE
		T_ExchgParam.T_FunctionCommon.xWarmUp_ContactorMachine_Active:= FALSE;
		T_ExchgParam.T_FunctionCommon.TWarmUp_Para:=T_NovRam.T_Data.TWarmUp_Para;
		T_ExchgParam.T_FunctionCommon.xWarmUp_MessageWarning:=FALSE;
		T_ExchgParam.T_FunctionCommon.iWarmUp_ColourChange:=0;
		TONWarmUpChangeColour(IN:=FALSE);
	END_IF;

(* ConfirmStartWarmUp *)  (* SOA 20.02.2023 *)
	IF xConfirmStartWarmUp THEN
		CASE iStepAction OF
		(* check state *)
		1:	xTmp:=	TRUE;
			(* next step *)
			xStopWarmup:=FALSE;
			xStartUpConfirmed:=FALSE;
			IF xTmp THEN iStepAction:=10; ELSE iStepAction:=90; END_IF;
		(*Check for Valid Warmup TimeEntry*)
		10: 	IF xWarmUp_Stop THEN
			T_ExchgParam.T_Visu.T_Message.iState:=126;   (* Ungültige/Keine Zeiteingabe für Warmup gewählt *)
				TONDelayMessage(IN:=TRUE,PT:=T#3s);
				IF TONDelayMessage.Q THEN
					TONDelayMessage(IN:=FALSE);
					iStepAction:=90;
				END_IF;
			ELSE iStepAction:=20;
			END_IF;
		(* Display message to ask for confirmation *)
		20:	T_ExchgParam.T_FunctionCommon.xWarmUp_MessageWarning_2:=TRUE;
			iStepAction:=30;
		(* Set Value *)
		30:	IF RisingEdgeKeyPanel_Enter.Q THEN
				xStartUpConfirmed:=TRUE;
				iStepAction:=90;
			ELSIF RisingEdgeKeyPanel_Esc.Q THEN
					T_ExchgParam.T_Visu.T_Message.iState:=5; (* Warnung: Aktion abgebrochen ! *)
					T_ExchgParam.T_FunctionCommon.xWarmUp_MessageWarning_2:=FALSE;
					xStartUpConfirmed := FALSE;
					iStepAction:=90;
			END_IF;
		(* action done *)
		90:	T_Visu.T_CtrleAction.xDone:=TRUE;
			T_Visu.T_CtrleAction.xNotReady:=FALSE;
			T_Visu.T_CtrleAction.xErr:=FALSE;
			T_Visu.T_CtrleAction.udiErrorID:=0;
			T_ExchgParam.T_Visu.T_Message.iState:=0;
			xConfirmStartWarmUp:=FALSE;
			T_ExchgParam.T_FunctionCommon.xWarmUp_MessageWarning_2:=FALSE;
			xTmp:=FALSE;
		END_CASE
	END_IF

	IF NOT(xInitReadFirstTimeTimeStamp) THEN
		(* lesen der Windows Systemzeit *)
		fbGetSysTime(	NETID:= '',
						START:= TRUE,
						TMOUT:= T#2s);
		IF NOT(fbGetSysTime.BUSY) OR fbGetSysTime.ERR THEN
			xInitReadFirstTimeTimeStamp:=TRUE;
			TIMESTR:=fbGetSysTime.TIMESTR;
			fbGetSysTime(	NETID:= '',
							START:= FALSE,
							TMOUT:= T#2s);
			T_ExchgParam.T_TimeStamp:=TIMESTR;
		END_IF;
	ELSE
		(* Refreshen der Zeit alle 60 Sekunden *)
		fbGetSysTime(	NETID:= '',
						START:= xGetTime,
						TMOUT:= T#2s);
		IF xGetTime AND NOT(fbGetSysTime.BUSY) THEN
			TIMESTR:=fbGetSysTime.TIMESTR;
			T_ExchgParam.T_TimeStamp:=TIMESTR;
			xGetTime:=FALSE;
		END_IF;
		TONWaitGetTime(IN:=TRUE,PT:=T#60s);
		IF TONWaitGetTime.Q THEN
			TONWaitGetTime(IN:=FALSE);
			xGetTime:=TRUE;
		END_IF;
	END_IF;

	(* Activate all WarmUp Elements*)
	xHydraulicStuder := xMotorStuder := xCoolantStuder := xCoolantPumpExt := T_ExchgParam.T_FunctionCommon.xWarmUp_ContactorMachine_Active;
	xMoveTableStuderBW :=T_ExchgParam.T_StationCommon.T_AutoGeometryPara.xMoveTableStuderBW;

	(*Activate external Coolant Pump when Contactor is not activ *)
	IF NOT T_TwinSafeIn.IxContactorAuxContact THEN
		IF (T_Visu.T_PlcParam.dwActualPage = 141) THEN
			xCoolantPumpExt := T_ExchgParam.T_FunctionCommon.xWarmUp_ContactorMachine_Active;
		ELSE
			xCoolantPumpExt := TRUE;
		END_IF;
	ELSE
		xCoolantPumpExt := FALSE;
	END_IF;

	(* Reset / Initialisierung *)
	IF T_Visu.T_PlcParam.dwActualPage <> 141 OR NOT xSecurityKey OR T_TwinSafeIn.IxContactorAuxContact OR xStopWarmup OR xStopProcess OR
		 xAction_StopCycle (* OR xStopImmediatly*) OR RisingEdgeActionError.Q OR T_Visu.T_PlcParam.dwActualPage = 141 AND T_NovRAM.T_Ctrle.xExecute THEN
		xConfirmStartWarmUp:=xStartUpConfirmed:=xSaveValueWarmUp:=xReadyToStartNextTime:=xWarmuUp_Start:=FALSE;
		T_ExchgParam.T_FunctionCommon.xWarmUp_ContactorMachine_Active:=T_ExchgParam.T_FunctionCommon.xWarmUp_MessageWarning_2:= FALSE;
		T_ExchgParam.T_FunctionCommon.xWarmUp_MessageWarning := FALSE;
		xStopWarmup:=FALSE;
	END_IF;

(* SOA 12.01.2023  } *)


(************************************************************************************************************************************************************************)
(***************                                             end for the section for defined function of the visualisation interface                                                ********************)
(************************************************************************************************************************************************************************)
END_ACTION
ACTION VisuFunction_SpecialFunction:
(* CW / CCW *)
IF xCWCCW OR xCylBrake THEN
	(* Step stop axis *)
	CASE iStepAction OF
	(* check axis *)
	1:	IF xCWCCW THEN	QxGrindingSpindle_CCW:=NOT(QxGrindingSpindle_CCW);					END_IF
		IF xCylBrake THEN	QxGrindingSpindle_ReleaseBrake:=NOT(QxGrindingSpindle_ReleaseBrake);	END_IF
		iStepAction:=90;
	(* action done *)
	90:	T_Visu.T_CtrleAction.xDone:=TRUE;
		T_Visu.T_CtrleAction.xNotReady:=FALSE;
		T_Visu.T_CtrleAction.xErr:=FALSE;
		T_Visu.T_CtrleAction.udiErrorID:=0;
		xCWCCW:=FALSE;
		xCylBrake:=FALSE;
	END_CASE
END_IF
END_ACTION
ACTION VisuFunction_StationFunction:
(* Action Station Function *)
	IF xActivateStationFunction THEN;
		(* Step  function station  *)
		CASE iStepAction OF
		(* check station state *)
		1:	xTmp:=	T_Station.TControl.xEnd AND
					T_Station.TControl.xRdy AND
					NOT(T_Station.TControl.xStart) AND
					NOT(T_Station.TControl.xError) AND
					NOT(T_Station.TControl.xStop) AND
					( (T_Visu.ptrT_ExchgParam^.T_StationCommon.rNewToolRotationSpeed <> 0) OR (iTmpStationFunctionNr = 20)) ;
			(* next step *)
			IF xTmp THEN iStepAction:=20; ELSE iStepAction:=95; END_IF
			IF xTmp AND T_Station.TControl.xHardwareConfigError THEN iStepAction:=95; END_IF;
		(* determin function number *)
		20:	IF (iTmpStationFunctionNr = 2) THEN
				bStateMachine:=2;
				xSetStateMachine:=TRUE;
			END_IF;
			T_Station.TControl.iFunctNr:=iTmpStationFunctionNr;
			CASE T_Station.TControl.iFunctNr OF
			(* available function, activ function *)
			2,3:	CASE T_Station.TControl.iFunctNr OF
				2:	T_Station.THardware.TAxisToolLeft.T_CtrleSingle.lrVelocity:=T_Visu.ptrT_ExchgParam^.T_StationCommon.rNewToolRotationSpeed;
					T_Station.THardware.TAxisToolLeft.T_CtrleSingle.lrAcceleration:=T_NovRAM.T_Data.T_Standard.T_TeachINToolLeft.rAcceleration;
					T_Station.THardware.TAxisToolLeft.T_CtrleSingle.lrDecceleration:=T_NovRAM.T_Data.T_Standard.T_TeachINToolLeft.rDeceleration;
					T_Station.THardware.TAxisToolLeft.T_CtrleSingle.lrGearDivider:=10000;
					T_Station.THardware.TAxisToolLeft.T_CtrleSingle.lrGearFactor:=10000;

					IF xMicroRodActive THEN
						(* ToolCenter --> Slave of ToolLeft only by MicroRod *)
						T_Station.THardware.TAxisToolCenter.T_CtrleSingle.lrAcceleration:=T_NovRAM.T_Data.T_Standard.T_TeachINToolCenter.rAcceleration;
						T_Station.THardware.TAxisToolCenter.T_CtrleSingle.lrDecceleration:=T_NovRAM.T_Data.T_Standard.T_TeachINToolCenter.rDeceleration;
						T_Station.THardware.TAxisToolCenter.T_CtrleSingle.lrGearDivider:=INT_TO_LREAL(T_Station.T_WorkTool.iBaseGearDivider);
						T_Station.THardware.TAxisToolCenter.T_CtrleSingle.lrGearFactor:=(	INT_TO_LREAL(T_Station.T_WorkTool.iBaseGearDivider) /
																						(T_Station.THardware.TAxisToolLeft.T_CtrleSingle.lrGearRatio /
																						T_Station.THardware.TAxisToolCenter.T_CtrleSingle.lrGearRatio)) * -1.0;
						(* ToolRight --> Slave of ToolLeft by MicroWire or Slave of ToolRight by MicroRod *)
						T_Station.THardware.TAxisToolRight.T_CtrleSingle.lrAcceleration:=T_NovRAM.T_Data.T_Standard.T_TeachINToolRight.rAcceleration;
						T_Station.THardware.TAxisToolRight.T_CtrleSingle.lrDecceleration:=T_NovRAM.T_Data.T_Standard.T_TeachINToolRight.rDeceleration;
						T_Station.THardware.TAxisToolRight.T_CtrleSingle.lrGearDivider:=INT_TO_LREAL(T_Station.T_WorkTool.iBaseGearDivider);
						T_Station.THardware.TAxisToolRight.T_CtrleSingle.lrGearFactor:=	INT_TO_LREAL(T_Station.T_WorkTool.iBaseGearDivider) /
																						(T_Station.THardware.TAxisToolLeft.T_CtrleSingle.lrGearRatio /
																						T_Station.THardware.TAxisToolRight.T_CtrleSingle.lrGearRatio);
					END_IF;
					IF NOT(xMicroRodActive) THEN
						(* ToolRight --> Slave of ToolRight by MicroWire *)
						T_Station.THardware.TAxisToolFeeder.T_CtrleSingle.lrAcceleration:=T_NovRAM.T_Data.T_Standard.T_TeachINToolFeeder.rAcceleration;
						T_Station.THardware.TAxisToolFeeder.T_CtrleSingle.lrDecceleration:=T_NovRAM.T_Data.T_Standard.T_TeachINToolFeeder.rDeceleration;
						T_Station.THardware.TAxisToolFeeder.T_CtrleSingle.lrGearDivider:=INT_TO_LREAL(T_Station.T_WorkTool.iBaseGearDivider);
						T_Station.THardware.TAxisToolFeeder.T_CtrleSingle.lrGearFactor:=	(INT_TO_LREAL(T_Station.T_WorkTool.iBaseGearDivider) /
																						(T_Station.THardware.TAxisToolFeeder.T_CtrleSingle.lrGearRatio /
																						T_Station.THardware.TAxisToolRight.T_CtrleSingle.lrGearRatio)) * -1.0;

						(* ToolRight --> Slave of ToolLeft by MicroWire or Slave of ToolRight by MicroRod *)
						T_Station.THardware.TAxisToolRight.T_CtrleSingle.lrAcceleration:=T_NovRAM.T_Data.T_Standard.T_TeachINToolRight.rAcceleration;
						T_Station.THardware.TAxisToolRight.T_CtrleSingle.lrDecceleration:=T_NovRAM.T_Data.T_Standard.T_TeachINToolRight.rDeceleration;
						T_Station.THardware.TAxisToolRight.T_CtrleSingle.lrGearDivider:=INT_TO_LREAL(T_Station.T_WorkTool.iBaseGearDivider);
						T_Station.THardware.TAxisToolRight.T_CtrleSingle.lrGearFactor:=	(INT_TO_LREAL(T_Station.T_WorkTool.iBaseGearDivider) /
																						(T_Station.THardware.TAxisToolLeft.T_CtrleSingle.lrGearRatio /
																						T_Station.THardware.TAxisToolRight.T_CtrleSingle.lrGearRatio)) * -1.0;
					END_IF;
				END_CASE;
				T_Station.TControl.xStart:=TRUE;
				IF (T_Station.TControl.iFunctNr = 2) THEN
					(* Display message *)
					T_Visu.ptrT_ExchgParam^.T_Visu.T_Message.iState:=25;
				END_IF;
				(* next step *)
				iStepAction:=30;
			(* not available function *)
			20:	T_Station.TControl.xStart:=TRUE;
			T_Visu.ptrT_ExchgParam^.T_Visu.T_Message.iState:=2;
(*				T_Visu.ptrT_ExchgParam^.T_SafetyCtrl.bStateReferenceMaxToolLength:=2;*)
				bStateMachine:=2;
				xSetStateMachine:=TRUE;
			    	iStepAction:=30;
			1,4..19,21..99:		iStepAction:=95;
			END_CASE
			(* next step *)
			xStepActionDone:=FALSE;
		(* wait confirmation *)
		30:	IF NOT(xStepActionDone) THEN
			(* release execution *)
				T_Station.TControl.xStart:=FALSE;
				xStepActionDone:=TRUE;
			ELSE
				IF T_Station.TControl.xEnd THEN
				(* action done *)
					IF(iTmpStationFunctionNr = 20) THEN
						iStepAction:=50;
					ELSE
						iStepAction:=90;
					END_IF;
					xStepActionDone:=FALSE;
				ELSE 	IF T_Station.TControl.xError THEN
						(* action error *)
							iStepAction:=99;
							xStepActionDone:=FALSE;
						END_IF
				END_IF
			END_IF
		(* Save NovRam *)
		50:	T_NovRam.T_Data.T_Standard.T_MachineConfig.rConfigMaxToolLength:=T_Station.THardware.TAxisToolFeeder.T_LiveValue.lrActualPosition *0.1;
			T_NovRam.T_Data.T_Standard.T_MachineConfig.rConfigMaxToolLengthOriginal:=T_Station.THardware.TAxisToolFeeder.T_LiveValue.lrActualPosition *0.1;
			T_Station.xOverwriteMaxToolLength:=TRUE;
			T_NovRAM.T_Ctrle.xExecute:=TRUE;
			T_NovRAM.T_Ctrle.iFunction:=2;
			iStepAction:=60;
		60:	IF NOT(xStepActionDone) THEN
				xStepActionDone:=TRUE;
				T_NovRAM.T_Ctrle.xExecute:=FALSE;
			END_IF;
			IF T_NovRAM.T_Ctrle.xDone THEN
				T_Station.T_MachineConfig.rConfigMaxToolLength:=T_NovRAM.T_Data.T_Standard.T_MachineConfig.rConfigMaxToolLength;
				T_Station.xOverwriteMaxToolLength:=FALSE;
				xStepActionDone:=FALSE;
				iStepAction:=90;
			END_IF;
		(* action done *)
		90:	IF (iTmpStationFunctionNr = 3) THEN
				bStateMachine:=1;
				xSetStateMachine:=TRUE;
			END_IF;
			IF (iTmpStationFunctionNr = 20) THEN
				T_Visu.ptrT_ExchgParam^.T_StationCommon.rConfigMaxToolLength:=T_NovRAM.T_Data.T_Standard.T_MachineConfig.rConfigMaxToolLength;
				T_Visu.ptrT_ExchgParam^.T_StationCommon.rConfigMaxToolLengthOriginal:=T_NovRAM.T_Data.T_Standard.T_MachineConfig.rConfigMaxToolLength;
				T_Visu.ptrT_ExchgParam^.T_Visu.T_Message.iState:=1;
(*				T_Visu.ptrT_ExchgParam^.T_SafetyCtrl.bStateReferenceMaxToolLength:=1;*)
				bStateMachine:=1;
				xSetStateMachine:=TRUE;
			END_IF;
			T_Visu.T_CtrleAction.xDone:=TRUE;
			T_Visu.T_CtrleAction.xNotReady:=FALSE;
			T_Visu.T_CtrleAction.xErr:=FALSE;
			T_Visu.T_CtrleAction.udiErrorID:=0;
			xActivateStationFunction:=FALSE;
		(* Configuration Error *)
		91:	T_Visu.T_CtrleAction.xDone:=TRUE;
			T_Visu.T_CtrleAction.xNotReady:=FALSE;
			T_Visu.T_CtrleAction.xErr:=FALSE;
			T_Visu.T_CtrleAction.udiErrorID:=0;
			xActivateStationFunction:=FALSE;
		(* function not ready *)
		95:	TimerNotReady(IN:=TRUE);
			xActivateStationFunction:=FALSE;
		(* error *)
		99:	T_Visu.T_CtrleAction.xDone:=TRUE;
			T_Visu.T_CtrleAction.xNotReady:=FALSE;
			FBErrorMessage(	diErrorNr:=T_Station.TControl.diErrorNr,
							T_ErrorList:=T_ErrorList);
			T_Visu.ptrT_ExchgParam^.T_Visu.T_Message.sDynamicTextEnglish:=FBErrorMessage.sErrorTextEnglish;
			T_Visu.ptrT_ExchgParam^.T_Visu.T_Message.sDynamicTextDeutsch:=FBErrorMessage.sErrorTextDeutsch;
			T_Visu.ptrT_ExchgParam^.T_Visu.T_Message.sDynamicTextFrancais:=FBErrorMessage.sErrorTextFrancais;
			T_Visu.T_CtrleAction.xErr:=FALSE;
			T_Visu.T_CtrleAction.udiErrorID:=0;
			xActivateStationFunction:=FALSE;
		END_CASE
	END_IF;
END_ACTION

(* POU PRG_VISU_LAYER5/FB_VISU/FBQVIS_INITPAGE, ST *)
FUNCTION_BLOCK FBQVIS_INITPAGE
VAR_INPUT
END_VAR
VAR_OUTPUT
END_VAR
VAR_IN_OUT
	T_Visu:ST_QVIS;			(* data structure of the visualisation *)
END_VAR
VAR
(* pointer *)
	ptrConfigPage: POINTER TO ST_CONFIGPAGE;
(* variable *)
	iIndexPage:INT;
	iPageNumber:INT;
(* variable Tmp *)
	i:INT;
END_VAR
(****************************************************************************************************************************************************)
(***********                    This Functionblock init all the defined page in QVis for the hole page management                            ************)
(****************************************************************************************************************************************************)
(* init. index array *)
FOR i:=0 TO 999 DO
	T_Visu.T_PageIndex[i].iIndexConfigPage:=0;
END_FOR
(* init. Number Page *)
iPageNumber:=0;



Page_000_Start;
Page_001_BIOS;
Page_002_BIOS;
Page_010_Auto_Geometry1;
Page_011_Auto_Geometry2;
Page_020_Auto_Groove1;
Page_021_Auto_Groove2;
Page_030_Auto_Reference;
Page_040_Auto_Setup1;
Page_041_Auto_Setup2;
Page_050_Auto_Info1;
Page_051_Auto_Info2;
Page_060_Auto_ErrorList;

Page_110_Setup_ToolCalibration;
Page_120_Setup_ToolGeometry1;
Page_121_Setup_ToolGeometry2;
Page_130_Setup_Profile;
Page_140_Setup_Setup1;
Page_141_Setup_Setup2;
Page_150_Setup_Config;
Page_160_Setup_ErrorList;
Page_170_Setup_Parameter;

Page_210_WorkStation_Axis1;
Page_220_WorkStation_ToolTorque;
Page_230_WorkStation_ToolTension;
Page_260_WorkStation_ErrorList;
Page_270_WorkStation_Parameter1;

Page_310_WorkStation_Axis2;
Page_320_WorkStation_SettingUp;
Page_330_WorkStation_Reference;
Page_360_WorkStation_ErrorList;
Page_370_WorkStation_Parameter2;

